# B&R Automation Studio project AriesV2 (part 2)

- acp10err-en.txt (not shown)

### ArUser.typ
```iecst
(********************************************************************
 * COPYRIGHT -- Bernecker + Rainer
 ********************************************************************
 * Library: ArUser
 * File: ArUser.typ
 * Author: B+R
 ********************************************************************
 * Data types of library ArUser
 ********************************************************************)

 TYPE
	ArUserIdentType : STRUCT
		Handle			: UDINT;
		MagicNumber		: UDINT;
	END_STRUCT;

	ArUserAsyncInternalType : STRUCT
		FBStateCtx		: ArFBStateInternalType;
		AsyFuMaCtx		: ArFBAsyFuMaInternalType;
	END_STRUCT;

	ArUserInternalType : STRUCT
		FBStateCtx		: ArFBStateInternalType;
	END_STRUCT;

END_TYPE
```

### AsGuard.var
```iecst
(********************************************************************
 * COPYRIGHT -- Bernecker + Rainer
 ********************************************************************
 * Library: AsGuard
 * File: AsGuard.var
 * Author: B+R
 ********************************************************************
 * Local variables of library AsGuard
 ********************************************************************)

(* error area 37300 - 37349 for AsGuard reserved *)

VAR CONSTANT
	guardERR_NULLPOINTER				: UINT := 37300;	(*null pointer specified*)
	guardERR_GENERAL					: UINT := 37301;	(*general license error*)
	guardERR_BUFFERSIZE					: UINT := 37302;	(*buffer too small*)
	guardERR_MEMORY						: UINT := 37303;	(*memory error*)
	guardERR_NOT_STARTED				: UINT := 37304;	(*license manager not started*)
	guardERR_ACCESS						: UINT := 37305;	(*license access error*)
	guardERR_VIOLATION					: UINT := 37306;	(*license violation*)
	guardERR_SERVICE_VIOLATION 			: UINT := 37307;	(*service mode because of license violation*)
	guardERR_CREATE_UPDATE_CONTEXT		: UINT := 37308;	(*error creating update context*)
	guardERR_CREATE_CONTEXT_FILE		: UINT := 37309;	(*error creating update context file*)
	guardERR_EXECUTE_UPDATE				: UINT := 37310;	(*error executing license update*)
	guardERR_FILE_NOT_FOUND				: UINT := 37311;	(*file not found*)
	guardERR_LIC_NOT_INITIALIZED		: UINT := 37312;	(*license not initialized*)
	guardERR_TASK						: UINT := 37313;
	guardERR_DONGLE_NOT_FOUND			: UINT := 37314;	(*specified dongle not found*)
	guardERR_CONTEXT_SIZE				: UINT := 37315;	(*wrong context size*)
	guardERR_INVALID_PARAM				: UINT := 37316;	(*invalid parameter specified*)
	guardERR_UNAVAILABLE				: UINT := 37317;	(*function unavailable*)
	guardERR_DATA_SIZE					: UINT := 37321;	(*data size invalid*)
	guardERR_LICENSE_STATUS_UNKNOWN		: UINT := 37322;	(*license status currently unknown*)

	guardBR_FIRMCODE                    : UDINT := 101652;	(*B&R firmcode*)

	guardLIC_REACT_NONE					: DWORD := 16#00;	(*no reaction*)
	guardLIC_REACT_LOGBOOK				: DWORD := 16#01;	(*in case of license violation write a message into logbook*)
	guardLIC_REACT_BLINK_CPU_LED		: DWORD := 16#02;	(*in case of license violation blink User LED*)
	guardLIC_REACT_BOOT_SERVICE			: DWORD := 16#04;	(*in case of license violation during bootup start PLC in service mode*)
	guardLIC_REACT_SERVICE				: DWORD := 16#08;	(*in case of license violation restart PLC in service mode *)

	guardREGISTER_ALWAYS				: DWORD := 1;		(*register license always*)
	guardREGISTER_IF_AVAILABLE			: DWORD := 2;		(*register license only if available*)

	guardGENERAL_OP_TIME_COUNTER 		: UDINT := 1;		(*general operating time counter*)
	guardCUSTOMER_OP_TIME_COUNTER		: UDINT := 2;		(*customer operating time counter*)
END_VAR
```

### AsHost.typ
```iecst
(********************************************************************
 * COPYRIGHT -- Bernecker + Rainer
 ********************************************************************
 * Library: AsHost
 * File: AsHost.typ
 * Author: B+R
 ********************************************************************
 * Data types of library AsHost
 ********************************************************************)

TYPE
	ASHOST_LOCAL_OBJ : STRUCT			(*internal use*)
		StateMan		: UINT;
		ErrMan			: UINT;
		Init			: UDINT;
		END_STRUCT;
END_TYPE
```

### AsOpcUac.typ
```iecst
(********************************************************************
 * COPYRIGHT -- Bernecker + Rainer
 ********************************************************************
 * Library: AsOpcUac
 * File:    AsOpcUac.typ
 * Author:  B+R
 ********************************************************************
 * Data types of library AsOpcUac
 ********************************************************************)

 TYPE
    (* Message security modes *)
	UASecurityMsgMode :
	(
    	UASecurityMsgMode_BestAvailable 	:= 0,	(* Detects best available mode the server provides (may result in no security) 	*)
	  	UASecurityMsgMode_None          	:= 1,	(* No secure communication 														*)
	  	UASecurityMsgMode_Sign          	:= 2,	(* Messages are signed to verify peer authenticity 								*)
	  	UASecurityMsgMode_SignEncrypt   	:= 3	(* Messages are signed and encrypted 											*)
	);

	(* Security policies *)
  	UASecurityPolicy :
  	(
    	UASecurityPolicy_BestAvailable  	:= 0,	(* Detects best available policy the server provides (may result in no security)	*)
    	UASecurityPolicy_None           	:= 1,	(* No secure communication (Allowed only for security mode = none)					*)
    	UASecurityPolicy_Basic128Rsa15  	:= 2,	(* RSA-PKCS-#1-V1.5-SHA1/RSA-PKCS-#1-V1.5/128-512 bit, HMAC-SHA1/AES-128-CBC/16bit	*)
    	UASecurityPolicy_Basic256       	:= 3,	(* RSA-PKCS-#1-OAEP-SHA1/RSA-OAEP/128-512 bit, HMAC-SHA1//AES-256-CBC/32bit			*)
    	UASecurityPolicy_Basic256Sha256   	:= 4	(* ???																				*)
  	);

  	(* Transport profiles to select encoding and protocol *)
  	UATransportProfile :
  	(
    	UATP_UATcp             				:= 1,	(* UA Binary over TCP								*)
    	UATP_WSHttpBinary      				:= 2,	(* Binary over HTTP			Not supported by B&R	*)
    	UATP_WSHttpXmlOrBinary 				:= 3,	(* XML/Binary over HTTP		Not supported by B&R	*)
    	UATP_WSHttpXml         				:= 4	(* XML over HTTP			Not supported by B&R	*)
  	);

  	(* Authentication token type provided for logon *)
 	UAUserIdentityTokenTtype :
 	(
 		UAUITT_Anonymous					:= 0,	(* Logon anonymously					*)
 		UAUITT_Username						:= 1,	(* Logon with user name and password 	*)
 		UAUITT_x509							:= 2	(* Logon with user certificate			*)
 	);

	(* Node identifier type *)
	UAIdentifierType :
	(
		UAIdentifierType_String 			:= 1,	(* String			*)
		UAIdentifierType_Numeric 			:= 2,	(* Numeric value	*)
		UAIdentifierType_GUID 				:= 3,	(* GUID				*)
		UAIdentifierType_Opaque				:= 4	(* ByteString		*)
	);

	(* Deadband type for monitored item sampling *)
	UADeadbandType :
	(
		UADeadbandType_None 				:= 0,	(* No deadband, each value change is sampled						*)
		UADeadbandType_Absolute 			:= 1,	(* Absolute value to exceed from last sample to make new sample		*)
		UADeadbandType_Percent				:= 2	(* Percent of EURange to exceed from last sample to make new sample	*)
	);

	UANodeClass :
	(
		UANodeClass_None 					:= 0,
		UANodeClass_Object					:= 1,
		UANodeClass_Variable 				:= 2,
		UANodeClass_Method					:= 4,
		UANodeClass_ObjectType				:= 8,
		UANodeClass_VariableType			:= 16,
		UANodeClass_ReferenceType			:= 32,
		UANodeClass_DataType				:= 64,
		UANodeClass_View					:= 128,
		UANodeClass_All						:= 255
	);

	UAAttributeId :
	(
	  	UAAI_Default						:= 0,
		UAAI_NodeId							:= 1,
		UAAI_NodeClass						:= 2,
		UAAI_BrowseName						:= 3,
		UAAI_DisplayName					:= 4,
		UAAI_Description					:= 5,
		UAAI_WriteMask						:= 6,
		UAAI_UserWriteMask					:= 7,
		UAAI_IsAbstract						:= 8,
		UAAI_Symmetric						:= 9,
		UAAI_InverseName					:= 10,
		UAAI_ContainsNoLoops				:= 11,
		UAAI_EventNotifier					:= 12,
		UAAI_Value							:= 13,
		UAAI_DataType						:= 14,
		UAAI_ValueRank						:= 15,
		UAAI_ArrayDimensions				:= 16,
		UAAI_AccessLevel					:= 17,
		UAAI_UserAccessLevel				:= 18,
		UAAI_MinimumSamplingInterval		:= 19,
		UAAI_Historizing					:= 20,
		UAAI_Executable						:= 21,
		UAAI_UserExecutable					:= 22
	);

	UAConnectionStatus :
	(
		UACS_Connected						:= 0,
		UACS_ConnectionError				:= 1,
		UACS_Shutdown						:= 2
	);

	UAServerState :
	(
		UASS_Running						:= 0,
		UASS_Failed							:= 1,
		UASS_NoConfiguration				:= 2,
		UASS_Suspended						:= 3,
		UASS_Shutdown						:= 4,
		UASS_Test							:= 5,
		UASS_CommunicationFault				:= 6,
		UASS_Unknown              			:= 7
	);

	UAVariantType :
	(										(* Kind of the variant data *)
		UAVariantType_Null					:= 0,	(* No data *)
		UAVariantType_Boolean				:= 1,	(* Data in element Boolean *)
		UAVariantType_SByte					:= 2,	(* Data in element SByte *)
		UAVariantType_Byte					:= 3,	(* Data in element Byte *)
		UAVariantType_Int16					:= 4,	(* Data in element Int16 *)
		UAVariantType_UInt16				:= 5,	(* Data in element UInt16 *)
		UAVariantType_Int32					:= 6,	(* Data in element Int32 *)
		UAVariantType_UInt32				:= 7,	(* Data in element UInt32 *)
		UAVariantType_Int64					:= 8,	(* Data in element Int64 *)
		UAVariantType_UInt64				:= 9,	(* Data in element UInt64 *)
		UAVariantType_Float					:= 10,	(* Data in element Float *)
		UAVariantType_Double				:= 11,	(* Data in element Double *)
		UAVariantType_String				:= 12,	(* Data in element String *)
		UAVariantType_DateTime				:= 13,	(* Data in element DateTime *)
		UAVariantType_Guid					:= 14,	(* Guid data in element String *)
		UAVariantType_ByteString			:= 15,	(* Byte string in element String *)
		UAVariantType_XmlElement			:= 16,	(* XML data in element String *)
		UAVariantType_NodeId				:= 17,	(* Data in element NodeId *)
		UAVariantType_ExpandedNodeId		:= 18,	(* Data in element ExpandedNodeId *)
		UAVariantType_StatusCode			:= 19,	(* Status code in element UInt32 *)
		UAVariantType_QualifiedName			:= 20,	(* Data in element QualifiedName *)
		UAVariantType_LocalizedText			:= 21	(* Data in element LocalizedText *)
	);

   	UAUserIdentityToken : STRUCT
		UserIdentityTokenType	: UAUserIdentityTokenTtype;
		TokenParam1 			: STRING[255];
		TokenParam2				: STRING[255];
	END_STRUCT;

 	UASessionConnectInfo : STRUCT
 	  	SessionName   			: STRING[255];
 	  	ApplicationName   		: STRING[255];
 	  	SecurityMsgMode   		: UASecurityMsgMode;
    	SecurityPolicy   		: UASecurityPolicy;
		CertificateStore		: STRING[255];
		ClientCertificateName	: STRING[255];
		ServerUri				: STRING[255];
		CheckServerCertificate	: BOOL;
    	TransportProfile 		: UATransportProfile;
    	UserIdentityToken		: UAUserIdentityToken;
		VendorSpecificParameter	: STRING[255];
    	SessionTimeout   		: TIME;
    	MonitorConnection		: TIME;
    	LocaleIDs				: ARRAY[0..4] OF STRING[6];
	END_STRUCT;

	(* Node identifier used to address nodes on the server *)
  	UANodeID : STRUCT
		NamespaceIndex			: UINT;							(* Index of the namespace which contains the node			*)
		Identifier 				: STRING[255];					(* Node identifier according to the identifier types format *)
		IdentifierType			: UAIdentifierType; 			(* String, Numeric, GUID, ByteString						*)
	END_STRUCT;

	(* Settings for data item monitoring *)
	UAMonitoringSettings : STRUCT
		SamplingInterval		: TIME;							(* Time in ms 															*)
		DeadbandType			: UADeadbandType; 				(* Deadband type which applies to deadband value						*)
		Deadband				: REAL; 						(* Deadband value, semantics depending on DeadbandType 					*)
	END_STRUCT;

	(* Settings for data item monitoring *)
	UAMonitoringParameters : STRUCT
		SamplingInterval		: TIME;							(* Time in ms 															*)
		QueueSize				: UINT;							(* Size of the server sided queue to collect value changes				*)
		DiscardOldest			: BOOL;							(* True to discard oldest on queue overflow or newest otherwise			*)
		DeadbandType			: UADeadbandType; 				(* Deadband type which applies to deadband value						*)
		Deadband				: REAL; 						(* Deadband value, semantics depending on DeadbandType 					*)
	END_STRUCT;

	UALocalizedText : STRUCT
		Locale					: STRING[6];
		Text					: STRING[255];
	END_STRUCT;

	UANodeInfo : STRUCT
		AccessLevel 			: BYTE;
		ArrayDimension			: ARRAY[0..MAX_INDEX_ARRAYDIMENSION] OF UDINT;
		BrowseName				: STRING[255];
		ContainsNoLoops 		: BOOL;
		DataType				: UANodeID;
		Description				: UALocalizedText;
		DisplayName				: UALocalizedText;
		EventNotifier			: BYTE;
		Executable				: BOOL;
		Historizing				: BOOL;
		InverseName				: STRING[255];
		IsAbstract				: BOOL;
		MinimumSamplingInterval	: TIME;
		NodeClass				: UANodeClass;
		NodeID					: UANodeID;
		Symmetric				: BOOL;
		UserAccessLevel			: BYTE;
		UserExecutable			: BOOL;
		UserWriteMask			: UDINT;
		ValueRank				: DINT;
		WriteMask				: UDINT;
	END_STRUCT;

	UAIndexRange : STRUCT
		StartIndex				: UINT;
		EndIndex 				: UINT;
	END_STRUCT;

	UANodeAdditionalInfo : STRUCT
		AttributeId				: UAAttributeId;
		IndexRangeCount			: UINT;
		IndexRange 				: ARRAY[0..MAX_INDEX_INDEXRANGE] OF UAIndexRange;
	END_STRUCT;

	(* Method argument used to supply the input and receive the output argument values for method calls *)
	UAMethodArgument : STRUCT
		Name					: STRING[64];		(* Name of the method argument								*)
		Value					: STRING[255];		(* Source/Destination variable name for the argument value	*)
	END_STRUCT;

	UAExpandedNodeID : STRUCT 	(* Expanded node identfier type *)
		NodeId					: UANodeID;
		NamespaceUri			: STRING[255];
		ServerIndex				: UDINT;
	END_STRUCT;

	UAQualifiedName : STRUCT	(* Qualified name type *)
		NamespaceIndex			: UINT;
		Name					: STRING[255];
	END_STRUCT;

	UARelativePathElement : STRUCT
	    ReferenceTypeId			: UANodeID;
		IsInverse				: BOOL;
		IncludeSubTypes			: BOOL;
		TargetName				: UAQualifiedName;
	END_STRUCT;

	UARelativePath : STRUCT
	    NoOfElements			: DWORD;
		Elements				: ARRAY[0..MAX_INDEX_RELATIVEPATH] OF UARelativePathElement;
	END_STRUCT;

	UADataValue : STRUCT		(* Additional informations about data value *)
		Valid 					: BOOL;
		Reserved				: ARRAY[0..2]OF USINT;
		StatusCode				: UDINT;
		SourceTimestamp			: DATE_AND_TIME;
		ServerTimestamp			: DATE_AND_TIME;
	END_STRUCT;

	UAVariantData : STRUCT		(* Standard type for variant data *)
		VariantType				: UAVariantType;
		Boolean					: BOOL;
		SByte					: SINT;
		Byte					: USINT;
		Int16					: INT;
		UInt16					: UINT;
		Int32					: DINT;
		UInt32					: UDINT;
		Float					: REAL;
		Double					: LREAL;
		DateTime				: DATE_AND_TIME;
		String					: STRING[255];
		NodeId					: UANodeID;
		ExpandedNodeId			: UAExpandedNodeID;
		QualifiedName			: UAQualifiedName;
		LocalizedText			: UALocalizedText;
		DataValue				: UADataValue;
	END_STRUCT;

	UARange : STRUCT			(* Range for a value *)
		Low						: LREAL;
		High					: LREAL;
	END_STRUCT;

	UAEUInformation : STRUCT 	(* Information about the engineering units *)
		NamespaceUri			: STRING[255];
		UnitId					: DINT;
		DisplayName				: UALocalizedText;
		Description				: UALocalizedText;
	END_STRUCT;

	UATimeZoneData : STRUCT		(* Information about time zone *)
		TimeOffset				: INT;	(* Offset in minutes from UTC *)
		DaylightSaving			: BOOL;	(* Offset includes the DST *)
	END_STRUCT;

END_TYPE
```

### AsSafety.typ
```iecst
(********************************************************************
 * COPYRIGHT -- Bernecker + Rainer
 ********************************************************************
 * Library: AsSafety
 * File: AsSafety.typ
 * Author: B&R
 * Created: May 25, 2012
 ********************************************************************
 * Data types of library AsSafety
 ********************************************************************)

TYPE
	RemoteControlCmdTypeV1 : 	STRUCT  (*remote control command structure*)
		Version : UINT; (*used version*)
		Command : UINT; (*command*)
		Number : UINT; (*actual number*)
		Data : UINT; (*data*)
		Password : STRING[16]; (*password*)
		NewPassword : STRING[16]; (*new password*)
	END_STRUCT;
	DownloadCmdMaOpTypeV1 : 	STRUCT  (*machine options command structure*)
		Version : UINT; (*used version*)
		Password : STRING[16]; (*password*)
		UDID_Low : UDINT; (*UDID low from SafeLOGIC*)
		UDID_High : UINT; (*UDID high from SafeLOGIC*)
		Unlock : USINT; (*unlock data*)
		pDeviceListInput : UDINT; (*pointer to device list*)
		NumberDevicesInput : UINT; (*number of devices*)
		pMachineOptionsInput : UDINT; (*pointer to bit machine options*)
		pModuleFlagsInput : UDINT; (*pointer to module flags*)
		pAcknMachineOptions : UDINT; (*pointer to acknowledge information*)
		pDeviceListOutput : UDINT; (*pointer to device list from SafeLOGIC*)
		NumberDevicesOutput : UINT; (*number of devices from SafeLOGIC*)
		pMachineOptionsOutput : UDINT; (*pointer to bit machine options from SafeLOGIC*)
		pModuleFlagsOutput : UDINT; (*pointer to module flags from SafeLOGIC*)
	END_STRUCT;
	DownloadDeviceTypeV1 : 	STRUCT  (*safety device*)
		SADR : UINT; (*safety address*)
		UDID_Low : UDINT; (*UDID low*)
		UDID_High : UINT; (*UDID high*)
	END_STRUCT;
	ConfigurationDeviceTypeV1 : 	STRUCT  (*safety device from SafeLOGIC*)
		SADR : UINT; (*safety address*)
		UDID : ARRAY[0..5]OF USINT; (*UDID*)
	END_STRUCT;
	ConfigurationBitOptionsTypeV1 : 	STRUCT  (*bit machine options*)
		BitData : ARRAY[0..63]OF USINT; (*bit array*)
	END_STRUCT;
	ConfigurationModuleFlagsTypeV1 : 	STRUCT  (*module flags*)
		Optional : ARRAY[0..127]OF USINT; (*optional*)
		Startup : ARRAY[0..127]OF USINT; (*startup*)
		NotPresent : ARRAY[0..127]OF USINT; (*not present*)
	END_STRUCT;
	DownloadCmdExtMaOpTypeV1 : 	STRUCT  (*extended machine options command structure*)
		Version : UINT; (*used version*)
		Password : STRING[16]; (*password*)
		UDID_Low : UDINT; (*UDID low*)
		UDID_High : UINT; (*UDID high*)
		Unlock : USINT; (*unlock data*)
		pIntDataInput : UDINT; (*pointer to INT data*)
		NumberIntInput : UINT; (*number of INT channels*)
		pUintDataInput : UDINT; (*pointer to UINT data*)
		NumberUintInput : UINT; (*number of UINT channels*)
		pDintDataInput : UDINT; (*pointer to DINT data*)
		NumberDintInput : UINT; (*number of DINT channels*)
		pUdintDataInput : UDINT; (*pointer to UDINT data*)
		NumberUdintInput : UINT; (*number of UDINT channels*)
		pAcknMachineOptions : UDINT; (*pointer to acknowledge information*)
		pIntDataOutput : UDINT; (*pointer to INT data from SafeLOGIC*)
		NumberIntOutput : UINT; (*number of INT channels from SafeLOGIC*)
		pUintDataOutput : UDINT; (*pointer to UINT data from SafeLOGIC*)
		NumberUintOutput : UINT; (*number of UINT channels from SafeLOGIC*)
		pDintDataOutput : UDINT; (*pointer to DINT data from SafeLOGIC*)
		NumberDintOutput : UINT; (*number of DINT channels from SafeLOGIC*)
		pUdintDataOutput : UDINT; (*pointer to UDINT data from SafeLOGIC*)
		NumberUdintOutput : UINT; (*number of UDINT channels from SafeLOGIC*)
	END_STRUCT;
	ConfigurationIntOptionsTypeV1 : 	STRUCT  (*INT machine options*)
		ID : UINT; (*id*)
		Value : INT; (*value*)
	END_STRUCT;
	ConfigurationUintOptionsTypeV1 : 	STRUCT  (*UINT machine options*)
		ID : UINT; (*id*)
		Value : UINT; (*value*)
	END_STRUCT;
	ConfigurationDintOptionsTypeV1 : 	STRUCT  (*DINT machine options*)
		ID : UINT; (*id*)
		Value : DINT; (*value*)
	END_STRUCT;
	ConfigurationUdintOptionsTypeV1 : 	STRUCT  (*UDINT machine options*)
		ID : UINT; (*id*)
		Value : UDINT; (*value*)
	END_STRUCT;
	DownloadCmdTableTypeV1 : 	STRUCT  (*table command structure*)
		Version : UINT; (*used version*)
		Password : STRING[16]; (*password*)
		UDID_Low : UDINT; (*UDID low*)
		UDID_High : UINT; (*UDID high*)
		Unlock : USINT; (*unlock data*)
		pTableDataInput : UDINT; (*pointer to table data*)
		NumberTablesInput : UINT; (*number of tables*)
		pTableDataOutput : UDINT; (*pointer to table data from SafeLOGIC*)
		NumberTablesOutput : UINT; (*number of tables from SafeLOGIC*)
	END_STRUCT;
	DownloadCmdAddParaTypeV1 : 	STRUCT  (*additional paramater command structure*)
		Version : UINT; (*used version*)
		Password : STRING[16]; (*password*)
		UDID_Low : UDINT; (*UDID low*)
		UDID_High : UINT; (*UDID high*)
		Unlock : USINT; (*unlock data*)
		pParaListInput : UDINT; (*pointer to additional parameter data*)
		NumberParaSetsInput : UINT; (*number of parameter sets*)
		pParaDataOutput : UDINT; (*pointer to additional parameter data from SafeLOGIC*)
		NumberParaSetsOutput : UINT; (*number of parameter sets from SafeLOGIC*)
	END_STRUCT;
	DownloadTableTypeV1 : 	STRUCT  (*table data*)
		Device : STRING[80]; (*device for file*)
		File : STRING[80]; (*file name*)
	END_STRUCT;
	ConfigurationTableTypeV1 : 	STRUCT  (*table data from SafeLOGIC*)
		ID : UINT; (*table id*)
		Type : USINT; (*table type*)
		NumberOfCRCs : UINT; (*number of CRCs*)
		pCRCData : UDINT; (*pointer to CRC values*)
	END_STRUCT;
	DownloadAddParaTypeV1 : 	STRUCT  (*additional parameter data*)
		SADR : UINT; (*safety address*)
		ID : USINT; (*id*)
		pParaData : UDINT; (*pointer to additional parameter data*)
		Length : UDINT; (*length*)
		pAcknAddPara : UDINT; (*pointer to acknowledge information*)
	END_STRUCT;
	ConfigurationAddParaTypeV1 : 	STRUCT  (*additional parameter data from SafeLOGIC*)
		SADR : UINT; (*safety address*)
		ID : USINT; (*id*)
		pParaData : UDINT; (*pointer to additional parameter data*)
		Length : UDINT; (*length*)
		CRC : UDINT; (*CRC*)
		Timestamp : UDINT; (*timestamp*)
	END_STRUCT;
	DownloadCmdApplicationTypeV1 : 	STRUCT  (*application command structure*)
		Version : UINT; (*used version*)
		Password : STRING[16]; (*password*)
		UDID_Low : UDINT; (*UDID low*)
		UDID_High : UINT; (*UDID high*)
		ApplicationID : UINT; (*application id*)
		Device : STRING[80]; (*device for file*)
		File : STRING[80]; (*file name*)
		Unlock : USINT; (*unlock application*)
	END_STRUCT;
	ConfigurationCmdMaOpTypeV1 : 	STRUCT  (*machine options from SafeLOGIC command structure*)
		Version : UINT; (*used version*)
		Password : STRING[16]; (*password*)
		pDeviceListOutput : UDINT; (*pointer to device list from SafeLOGIC*)
		NumberDevicesOutput : UINT; (*number of devices from SafeLOGIC*)
		pMachineOptionsOutput : UDINT; (*pointer to bit machine options from SafeLOGIC*)
		pModuleFlagsOutput : UDINT; (*pointer to module flags from SafeLOGIC*)
	END_STRUCT;
	ConfigurationCmdExtMaOpTypeV1 : 	STRUCT  (*extended machine options from SafeLOGIC command structure*)
		Version : UINT; (*used version*)
		Password : STRING[16]; (*password*)
		pIntDataOutput : UDINT; (*pointer to INT data from SafeLOGIC*)
		NumberIntOutput : UINT; (*number of INT channels from SafeLOGIC*)
		pUintDataOutput : UDINT; (*pointer to UINT data from SafeLOGIC*)
		NumberUintOutput : UINT; (*number of UINT channels from SafeLOGIC*)
		pDintDataOutput : UDINT; (*pointer to DINT data from SafeLOGIC*)
		NumberDintOutput : UINT; (*number of DINT channels from SafeLOGIC*)
		pUdintDataOutput : UDINT; (*pointer to UDINT data from SafeLOGIC*)
		NumberUdintOutput : UINT; (*number of UDINT channels from SafeLOGIC*)
	END_STRUCT;
	ConfigurationCmdTableTypeV1 : 	STRUCT  (*table data from SafeLOGIC command structure*)
		Version : UINT; (*used version*)
		Password : STRING[16]; (*password*)
		pTableDataOutput : UDINT; (*pointer to table data from SafeLOGIC*)
		NumberTablesOutput : UINT; (*number of tables from SafeLOGIC*)
	END_STRUCT;
	ConfigurationCmdAddParaTypeV1 : 	STRUCT  (*additional parameter data from SafeLOGIC command structure*)
		Version : UINT; (*used version*)
		Password : STRING[16]; (*password*)
		pParaDataOutput : UDINT; (*pointer to additional parameter data from SafeLOGIC*)
		NumberParaSetsOutput : UINT; (*number of parameter sets from SafeLOGIC*)
	END_STRUCT;
	RemoteControlStatusTypeV1 : 	STRUCT  (*remote control status from SafeLOGIC*)
		Command : UINT; (*last received command*)
		Number : UINT; (*running number of last received command*)
		Status : UINT; (*status of command*)
		State : UINT; (*state of the last ENTER command*)
		EnterData : UINT; (*last received ENTER command that was correct executed*)
		EnterNumber : UINT; (*running number of the last received ENTER command*)
		EnterExecuteStatus : UINT; (*state of the last received ENTER command*)
		SafeOSState : USINT; (*status of the safety application*)
		SafeKEYChanged : USINT; (*SafeKEY has been exchanged*)
		LedTestActive : USINT; (*LED test active*)
		Scanning : USINT; (*module scan active*)
		openSAFETYstate : USINT; (*status of openSAFETY stack*)
		FailSafe : USINT; (*Fail-Safe status*)
		NumberOfMissingModules : UINT; (*number of missing modules*)
		NumberOfUDIDMismatches : UINT; (*number of mismatched modules*)
		NumberOfDifferentFirmware : UINT; (*number of modules with different firmware*)
		SADR : ARRAY[0..100]OF UINT; (*safety address array*)
		MissingModules : ARRAY[0..15]OF USINT; (*missing modules array*)
		UDIDMismatches : ARRAY[0..15]OF USINT; (*udid mismatch array*)
		DifferentFirmware : ARRAY[0..15]OF USINT; (*different firmware array*)
	END_STRUCT;
	DownloadAcknMaOpTypeV1 : 	STRUCT  (*acknowledge bit machine options structure*)
		AcknBitOptions : ARRAY[0..63]OF USINT; (*acknowledge bit*)
	END_STRUCT;
	DownloadAcknAddParaTypeV1 : 	STRUCT  (*acknowledge bit additional parameter*)
		AcknBitAddPara : ARRAY[0..63]OF USINT; (*acknowledge bit*)
	END_STRUCT;
	DownloadAcknExtMaOpTypeV1 : 	STRUCT  (*acknowledge extended machine options structure*)
		AcknIntOptions : ARRAY[0..63]OF BOOL; (*acknowledge INT*)
		AcknUintOptions : ARRAY[0..63]OF BOOL; (*acknowledge UINT*)
		AcknDintOptions : ARRAY[0..63]OF BOOL; (*acknowledge DINT*)
		AcknUdintOptions : ARRAY[0..63]OF BOOL; (*acknowledge UDINT*)
	END_STRUCT;
END_TYPE
```

### AsSafety.var
```iecst
(********************************************************************
 * COPYRIGHT -- Bernecker + Rainer
 ********************************************************************
 * Library: AsSafety
 * File: AsSafety.var
 * Author: B&R
 * Created: May 25, 2012
 ********************************************************************
 * Constants of library AsSafety
 ********************************************************************)
VAR CONSTANT
	safeVERSION_R107 : UINT := 16#107; (*safety release version - for 1.7 or higher*)
	safeDATA_TYPE_MAOP : UINT := 16#100; (*download type for machine options *)
	safeDATA_TYPE_EXTMAOP : UINT := 16#200; (*download type for extended machine options *)
	safeDATA_TYPE_TABLE : UINT := 16#300; (*download type for table objects *)
	safeDATA_TYPE_ADDPARA : UINT := 16#400; (*download type for additional parameter*)
	safeCMD_ENTER : UINT := 16#100; (*enter command*)
	safeCMD_STATUS : UINT := 16#200; (*status command*)
	safeCMD_STATUS_SL : UINT := 16#0000; (*read back status*)
	safeCMD_N_UDID_ACKN : UINT := 16#20; (*acknowledge N modules*)
	safeCMD_4_UDID_ACKN : UINT := 16#30; (*acknowledge 4 modules*)
	safeCMD_3_UDID_ACKN : UINT := 16#40; (*acknowledge 3 modules*)
	safeCMD_2_UDID_ACKN : UINT := 16#50; (*acknowledge 2 modules*)
	safeCMD_1_UDID_ACKN : UINT := 16#60; (*acknowledge 1 module*)
	safeCMD_FW_ACKN : UINT := 16#100; (*acknowledge firmware*)
	safeCMD_SK_XCHG : UINT := 16#200; (*acknowledge SafeKEY*)
	safeCMD_TEST : UINT := 16#1000; (*LED test*)
	safeCMD_SCAN : UINT := 16#2000; (*scan*)
	safeCMD_SK_PW : UINT := 16#5000; (*change password*)
	safeCMD_SK_FORMAT : UINT := 16#6000; (*format SafeKEY*)
	safeCMD_RESET : UINT := 16#7000; (*reset SafeLOGIC*)
	safeCMD_CLEAR_DATA : UINT := 16#8000; (*clear additonal downloaded data*)
	safeERR_VERSION : UINT := 36100; (*error wrong version for command structure*)
	safeERR_PW_LENGTH : UINT := 36101; (*error wrong password length*)
	safeERR_UDID : UINT := 36102; (*error no UDID*)
	safeERR_ALLOC_MEM : UINT := 36103; (*error allocating memory*)
	safeERR_INTERNAL_ERROR : UINT := 36104; (*internal error*)
	safeERR_TIMEOUT : UINT := 36105; (*error connection timeout*)
	safeERR_RC_CMD : UINT := 36106; (*error wrong command*)
	safeERR_RC_ENTER_DATA : UINT := 36107; (*error wrong data for ENTER command*)
	safeERR_RC_ENTER_PW : UINT := 36108; (*error no password for command*)
	safeERR_RC_ENTER_SK_PW : UINT := 36109; (*error no new password for command*)
	safeERR_RC_STATUS_DATA : UINT := 36110; (*error wrong data for STATUS command*)
	safeERR_RC_DATA_LENGTH : UINT := 36111; (*error worng length for status data*)
	safeERR_DL_NO_PASSWORD : UINT := 36112; (*error no password for download*)
	safeERR_DL_PROTOCOL : UINT := 36113; (*error protocol version for download*)
	safeERR_DL_FILE_OPEN : UINT := 36114; (*error file open*)
	safeERR_DL_FILE_INVALID : UINT := 36115; (*error file invalid*)
	safeERR_DL_FILE_TOO_BIG : UINT := 36116; (*error file too big*)
	safeERR_DL_WRITE : UINT := 36117; (*error write*)
	safeERR_DL_STREAM : UINT := 36118; (*error stream*)
	safeERR_DL_CHECKSUM : UINT := 36119; (*error checksum*)
	safeERR_DL_UDID : UINT := 36120; (*error UDID doesn't match*)
	safeERR_DL_WRONG_FILE_SIZE : UINT := 36121; (*error wrong file size*)
	safeERR_DL_NO_RIGHTS_TO_WRITE : UINT := 36122; (*error wrong password*)
	safeERR_DL_UNLOCK_FILE_INFO : UINT := 36123; (*error file info*)
	safeERR_DL_UNLOCK_READ : UINT := 36124; (*error unlock read*)
	safeERR_DL_UNLOCK_WRITE : UINT := 36125; (*error unlock write*)
	safeERR_DL_STATIC_UNLOCK : UINT := 36126; (*error static unlock*)
	safeERR_DL_COMPARE_FAILED : UINT := 36127; (*error data compare failed*)
	safeERR_DLDATA_TYPE_ERR : UINT := 36128; (*error data type for download*)
	safeERR_DLDATA_ERR_DATA : UINT := 36129; (*error data for download*)
	safeERR_COT_TYPE_ERR : UINT := 36130; (*error data type for upload*)
	safeERR_COT_READING_FILE : UINT := 36131; (*error reading file*)
END_VAR
```

### GmcManager.typ
```iecst
TYPE
	(*Enum types*)

	MCBufferModeEnum :
	(
		mcABORTING, (*Default mode with no buffering. The function block aborts an active movement. The buffer is cleared.*)
		mcBUFFERED 	(*The movement is started as soon as the previous movement is completed. No smoothing is applied.*)
	);

	MCCoordinateSystemEnum :
	(
		mcACS := 0,	(*Axis coordinate system*)
		mcMCS := 1,	(*Machine coordinate system*)
		mcPCS := 2,	(*Product coordinate system*)
		mcSCS1 := 3,	(*System coordinate system 1*)
		mcSCS2 := 4,	(*System coordinate system 2*)
		mcSCS3 := 5,	(*System coordinate system 3*)
		mcSCS4 := 6,	(*System coordinate system 4*)
		mcSCS5 := 7,	(*System coordinate system 5*)
		mcJACS := 100	(*Joint axis coordinate system*)
	);

	MCDirectionEnum :
	(
		mcDIR_POSITIVE,	(*positive direction*)
		mcDIR_NEGATIVE,	(*negative direction*)
		mcDIR_CURRENT,	(*current direction*)
		mcDIR_SHORTEST_WAY,		(*shortest way*)
		mcDIR_EXCEED_PERIOD := 8,	(*exceed period*)
		mcDIR_UNDEFINED	(*undefined direction*)
	);

	MCErrorCommandEnum :
	(
		mcWARNING_CMD := 0, (*a warning is generated*)
		mcERROR_CMD, (*Generates an error*)
		mcERROR_STOP_CMD, (*Generates an error and stops.*)
		mcERROR_STOP_CTRL_OFF_CMD, (*an axis error is generated on the drive, any active movement is aborted and the controller is switched off*)
		mcERROR_V_STOP_CTRL_OFF_CMD (*an axis error is generated on the drive, any active movement is ended with a speed ramp and controller is switched off*)
	);

	MCExecutionModeEnum :
	(
		mcEM_IMMEDIATELY,	(*The function is executed immediately.*)
		mcEM_QUEUED			(*The function is executed with a buffer.*)
	);

	MCGroupOperationModeEnum :
	(
		mcOM_M1_STOP, (*Optional stop*)
		mcOM_FEED_FORWARD, (*Feed forward*)
		mcOM_OPTMOT, (*Jerk-limiting trajectory planner*)
		mcOM_SAVE_RESTARTDATA (*Save data to restart a program*)
	);

	MCUnloadProgramModeEnum :
	(
		mcUPRG_NAME, (*Unload program by name*)
		mcUPGR_ALL (*Unload all programs*)
	);

	MCHomingModeEnum :
	(
		mcHOMING_DIRECT := 0,			(*Direct homing*)
		mcHOMING_SWITCH_GATE,			(*Homing with reference gate*)
		mcHOMING_ABSOLUTE_SWITCH,		(*Performs homing with absolute reference switch*)
		mcHOMING_LIMIT_SWITCH := 4,	    (*Homing with hardware limit switch*)
		mcHOMING_ABSOLUTE,				(*Homing by setting the homing offset*)
		mcHOMING_DCM := 7,				(*Homing using interval-encoded reference marks*)
		mcHOMING_BLOCK_TORQUE := 9,	    (*Performs homing to mechanical limit, torque as criteria*)
		mcHOMING_BLOCK_LAG_ERROR := 10,	(*Performs homing to mechanical limit, lag error as criteria*)
		mcHOMING_ABSOLUTE_CORRECTION := 133, (*Homing by setting the homing offset with counting range correction*)
		mcHOMING_DCM_CORRECTION := 135,	(*Homing using distance-coded reference marks with counting range correction*)
		mcHOMING_DEFAULT := 140,		(*Applies all parameters from the configuration*)
		mcHOMING_INIT,					(*init*)
		mcHOMING_RESTORE_POSITION		(*Restores position from permanent memory*)
	);

	MCHomingOrderSourceEnum :
	(
		mcHO_CONFIGURATION := 0,	(*Uses the homing order configured in the configuration*)
		mcHO_FUNCTIONBLOCK			(*Uses the homing order configured in the function block*)
	);

	MCInterpolationModeEnum :
	(
		mcIPLM_OFF,						(*interpolation off*)
		mcIPLM_LINEAR,					(*linear interpolation*)
		mcIPLM_QUADRATIC,				(*quadratic interpolation*)
		mcIPLM_QUADRATIC_NO_OVERSHOOT	(*quadratic interpolation without overshoot*)
	);

	MCOverrideEnum :
	(
		mcOVERRIDE_VELOCITY,			(*Speed override*)
		mcOVERRIDE_VELOCITY_AXIS,		(*Axis speed override*)
		mcOVERRIDE_ACCELERATION,		(*Acceleration override*)
		mcOVERRIDE_ACCELERATION_AXIS,	(*Axis acceleration override*)
		mcOVERRIDE_JERK,				(*Jerk override*)
		mcOVERRIDE_FEEDRATE := 10,		(*Feed override*)
		mcOVERRIDE_RAPID,				(*Rapid motion override*)
		mcOVERRIDE_SPINDLE,				(*Spindle override*)
		mcOVERRIDE_TIMESTRETCH := 20	(*Time stretch override*)
	);

	MCPlcopenParameterEnum :
	(
		mcPAR_COMMANDED_AX_POSITION := 1, 	(*Commanded position*)
		mcPAR_SW_LIMIT_POSITIVE,		(*Positive software limit*)
		mcPAR_SW_LIMIT_NEGATIVE,		(*Negative software limit*)
		mcPAR_ENABLE_LIMIT_POSITIVE,	(*Enable positive software limit switch*)
		mcPAR_ENABLE_LIMIT_NEGATIVE,	(*Enable negative software limit switch*)
		mcPAR_ENABLE_POS_LAG_MONITORING,	(*Enable monitoring of position lag*)
		mcPAR_MAX_AX_POSITION_LAG,		(*Maximum position lag*)
		mcPAR_MAX_AX_VELOCITY_SYSTEM,	(*Maximum velocity of the axis in the system*)
		mcPAR_MAX_AX_VELOCITY_APPL,		(*Maximum velocity of the axis in the application*)
		mcPAR_ACTUAL_AX_VELOCITY,  		(*Actual velocity of the axis*)
		mcPAR_COMMANDED_AX_VELOCITY,	(*Commanded velocity*)
		mcPAR_MAX_AX_ACCELERATION_SYSTEM,	(*Maximum acceleration of the axis in the system*)
		mcPAR_MAX_AX_ACCELERATION_APPL,	(*Maximum acceleration of the axis in the application*)
		mcPAR_MAX_AX_DECELERATION_SYSTEM,	(*Maximum deceleration of the axis in the system*)
		mcPAR_MAX_AX_DECELERATION_APPL,	(*Maximum deceleration of the axis in the application*)
		mcPAR_MAX_AX_JERK,			(*Maximum jerk of the axis*)
		mcPAR_AX_PERIOD := 1008,    (*Period of the axis*)
		mcPAR_HOMING_OFFSET := 1019, 	(*Homing offset of the axis*)
		mcPAR_AX_MEASUREMENT_RESOLUTION := 1020  (*Measurement resolution of the axis*)
	);

	MCNetworkTypeEnum :
	(
		mcNETWORK_POWERLINK	(*ETHERNET POWERLINK protocol*)
	);

	MCPrgAxesReposTypeEnum :
	(
		mcPRGRP_SINGLE_AXIS,			(*Single axis*)
		mcPRGRP_PROGRAM,				(*Program*)
		mcPRGRP_SINGLE_AXIS_AUTOMATIC	(*Single axis automatic*)
	);

	MCPrgInfoInterruptEnum :
	(
		mcINTERRUPT_NOT_INTERRUPTED,	(*The program has not been interrupted.*)
		mcINTERRUPT_SINGLESTEP,			(*The program has been interrupted by activation of single-step mode.*)
		mcINTERRUPT_FB,					(*The program has been interrupted by the "MC_GroupInterrupt" function block.*)
		mcINTERRUPT_INTERPRETER,		(*The program has been interrupted by an interpreter halt (G170).*)
		mcINTERRUPT_MFUNCTION,			(*The program has been interrupted by a blocking M-code.*)
		mcINTERRUPT_PROGRAM				(*The program has been interrupted by a programmed command.*)
	);

	MCPrgInfoModeEnum :
	(
		mcPRGIM_LIVE,		(*Live data*)
		mcPRGIM_ABORT_POINT (*Abortpoint data*)
	);

	MCRestartModeEnum :
	(
	   	mcRSM_ABORT_LINE,		(*Restart at abort line*)
		mcRSM_PATH_DISTANCE,	(*Restart at path distance*)
		mcRSM_BLOCK_NUMBER,		(*Restart at block number*)
		mcRSM_LINE_NUMBER,		(*Restart at line number*)
		mcRSM_TOOL_NUMBER,		(*Restart at tool number*)
		mcRSM_LABEL				(*Restart at label*)
	);

	MCRestartPhaseEnum :
	(
		mcRSP_INACTIVE,
		mcRSP_VALIDATE_PLAY_BACK_DATA,
		mcRSP_WAIT_START_AXES_REPOS,
		mcRSP_AXES_REPOSITIONING,
		mcRSP_WAIT_RESTART_PROGRAM,
		mcRSP_RUN_PROGRAM,
		mcRSP_PROGRAM_FINISHED
	);

	MCPrgStartModeEnum :
	(
		mcPRGSM_NON_MODAL,		(*Non Modal*)
		mcPRGSM_MODAL,		(*Modal*)
		mcPRGSM_RESTART		(*Restart*)
	);

	MCPrgStartPointEnum :
	(
		mcPRGSP_STANDARD,		(*Standard*)
		mcPRGSP_BLOCK_NUMBER,	(*Block Number*)
		mcPRGSP_ABORT_LINE,	(*Abort Line*)
		mcPRGSP_ABORT_POINT,	(*Abort Point*)
		mcPRGSP_PATH_DISTANCE,	(*Path Distance*)
		mcPRGSP_LINE_NUMBER	(*Line Number*)
	);

	MCPrgPhaseEnum :
	(
		mcPRGPH_INACTIVE,					(*Inactive*)
		mcPRGPH_SIMULATION_RUN,			(*Simulation run is active*)
		mcPRGPH_WAIT_FOR_AXES_REPOS,		(*Waiting for axes repositioning*)
		mcPRGPH_AXES_REPOS,				(*Axes repositioning is active*)
		mcPRGPH_WAIT_FOR_REAL_RUN,			(*Waiting for real run*)
		mcPRGPH_REAL_RUN					(*Real run is active*)
	);

	MCSimulationCommandEnum :
	(
		mcSIMULATION_SW_OFF,	(*simulation off*)
		mcSIMULATION_SW_ON		(*motor simulation*)
	);

	MCSwitchEnum :
	(
		mcSWITCH_STATE_OFF,		(*off*)
		mcSWITCH_STATE_ON		(*on*)
	);

	MCTransitionModeEnum :
	(
		mcTM_NONE		(*No transition is applied*)
	);

	MCValueSourceEnum :
	(
		mcVALUE_SET, 					(*Set position is used*)
		mcVALUE_ACTUAL,					(*Actual position is used*)
		mcVALUE_SET_AXIS_UNITS,			(*Set position in axis units is used*)
		mcVALUE_ACTUAL_AXIS_UNITS,		(*Actual position in axis units is used*)
		mcVALUE_AUTOMATIC_SELECTION			(*Mode only for ReadCyclicPosition: use the value depending on the ctrl mode*)
	);

	MCEdgeEnum :
	(
		mcEDGE_POSITIVE,				(*change from logical low to logical high*)
		mcEDGE_NEGATIVE					(*change from logical high to logical low*)
	);

	MCBrakeCommandEnum :
	(
		mcBRAKE_CLOSE,					(*close brake*)
		mcBRAKE_OPEN,					(*open brake*)
		mcBRAKE_GET_STATUS				(*show status of brake*)
	);

	MCBrakeStatusEnum :
	(
		mcBRAKE_STATUS_NOT_PROVIDED,			(*command was not mcBRAKE_GET_STATUS*)
		mcBRAKE_CLOSED,					(*holding brake closed*)
		mcBRAKE_OPENED					(*holding brake open*)
	);

	MCSegmentProcessParIDModeEnum :
	(
		mcSEG_PARID_GET := 0, (*read ParID once from the segment*)
		mcSEG_PARID_SET	(*write ParID once to the segment*)
	);

	MCSegmentDataTypeEnum :
		(
		mcSEG_PARTYPE_BOOL := 1, (*data type BOOL*)
		mcSEG_PARTYPE_SINT, (*data type SINT*)
		mcSEG_PARTYPE_INT, (*data type INT*)
		mcSEG_PARTYPE_DINT, (*data type DINT*)
		mcSEG_PARTYPE_USINT, (*data type USINT*)
		mcSEG_PARTYPE_UINT, (*data type UINT*)
		mcSEG_PARTYPE_UDINT, (*data type UDINT*)
		mcSEG_PARTYPE_REAL, (*data type REAL*)
		mcSEG_PARTYPE_VOID := 65535  (*data type unknown*)
	);

	(*Structure types*)

	MCAdditionalGroupHome_15_Type : STRUCT
		HomingOrderSource : MCHomingOrderSourceEnum;	(*Source of the homing order*)
    	HomingOrder : ARRAY[0..14] OF UINT;				(*Specifies the homing order (see HomingOrder) The array is in ACS order.*)
	END_STRUCT;

	MCAdditionalStatusType : STRUCT
		TriggerSwitch1 : BOOL;
		TriggerSwitch2 : BOOL;
		DriveEnableSwitch : BOOL;
		ResetDone : BOOL;
		LagWarning : BOOL;
	END_STRUCT;

	MCAdvancedMoveCycParType : STRUCT
		Velocity : REAL;
		Acceleration : REAL;
		Deceleration : REAL;
		DisableJoltLimitation : BOOL;
	END_STRUCT;

	MCAdvancedVelCtrlParType : STRUCT
		Acceleration : REAL;
		Deceleration : REAL;
	END_STRUCT;

	MCAdvancedGearInParType : STRUCT
		MasterMaxVelocity : REAL;
	END_STRUCT;

	MCCamTableDefineType : STRUCT
		DataObjectName : STRING[12];
		DataAdress : UDINT;
	END_STRUCT;

	MCFrameOrientationType : STRUCT
		Type : UDINT;		(*Describes the representation of rotation angles 1 to 3*)
		Angle1 : LREAL;		(*Rotation angle 1 for describing the orientation*)
		Angle2 : LREAL;		(*Rotation angle 2 for describing the orientation*)
		Angle3 : LREAL;		(*Rotation angle 3 for describing the orientation*)
	END_STRUCT;

	MCFramePositionType : STRUCT
		X : LREAL;		(*Offset in the direction of the X-axis*)
		Y : LREAL;		(*Offset in the direction of the Y-axis*)
		Z : LREAL;		(*Offset in the direction of the Z-axis*)
	END_STRUCT;

	MCFrameType : STRUCT
		Trans : MCFramePositionType;	(*Position*)
		Rot : MCFrameOrientationType;	(*Orientation*)
	END_STRUCT;

	MCKinematicTrfType : UDINT;

	MCPrgInfoActiveProgramType : STRUCT 		(*Informations about the active program*)
		Name : STRING[260];						(*Name of the active program*)
		Number : UDINT;							(*Number of the active program*)
		Level : UINT;							(*Current program level*)
	END_STRUCT;

	MCPrgInfoBlockMonType : STRUCT (*Block monitor*)
		LineNumber : UDINT;				(*Current line number*)
		BlockNumber : UDINT;			(*Current block number*)
		LineLast2 : STRING[260];		(*Second to last line in the sequence program*)
		LineLast1 : STRING[260];		(*Last line in the sequence program*)
		LineActual : STRING[260];		(*Current line in the sequence program*)
		LineNext1 : STRING[260];		(*Next line in the sequence program*)
		LineNext2 : STRING[260];		(*Line following the next line in the sequence program*)
		RemainingDistance : LREAL;		(*Distance remaining until the end of the block [units]*)
		Length : LREAL;					(*Length of the path of the current block [units]*)
		LengthNext : LREAL;				(*Length of the path of the next block [units]*)
	END_STRUCT;

	MCPrgInfoPrgHierarchyLevelType : STRUCT  (*Program Hierarchy Levels*)
		LineNumber : UDINT;				(*Current level line number*)
	END_STRUCT;

	MCPrgInfoPrgHierarchyType : STRUCT (*Program Hierarchy*)
		Level : ARRAY[0..14] OF MCPrgInfoPrgHierarchyLevelType; (*Program Hierarchy Levels*)
	END_STRUCT;

	MCPrgInfoAxesMonType : STRUCT (*Axes Monitor*)
		Position : ARRAY[0..14] OF LREAL; (*Axes positions*)
	END_STRUCT;

	MCPrgInfoType : STRUCT (*The structure contains extended information about the running program*)
		InitProgram : STRING[260];						(*Name of the initialization subroutine*)
		ActiveProgram : MCPrgInfoActiveProgramType;		(*Information about the active program*)
		InterruptStatus : MCPrgInfoInterruptEnum;		(*Interrupt informations*)
		BlockMonitor : MCPrgInfoBlockMonType;			(*Block monitor*)
		ProgramHierarchy : MCPrgInfoPrgHierarchyType;	(*Program Hierarchy*)
	END_STRUCT;

	MCPrgInfo15Type : STRUCT (*The structure contains extended information about the running program*)
		InitProgram : STRING[260];						(*Name of the initialization subroutine*)
		ActiveProgram : MCPrgInfoActiveProgramType;		(*Information about the active program*)
		InterruptStatus : MCPrgInfoInterruptEnum;		(*Interrupt informations*)
		BlockMonitor : MCPrgInfoBlockMonType;			(*Block monitor*)
		ProgramHierarchy : MCPrgInfoPrgHierarchyType;	(*Program Hierarchy*)
		AxesMonitor : MCPrgInfoAxesMonType; 			(*Axes monitor*)
	END_STRUCT;

	MCPrgInfoParAxesMonType : STRUCT (*The structure contains parameters for the axes monitor*)
		CoordSystem : MCCoordinateSystemEnum; (*Define order of monitored axes*)
	END_STRUCT;

	MCPrgInfoParType : STRUCT (*The structure contains parameters for the program informations*)
		Mode : MCPrgInfoModeEnum; (*Source of monitored data*)
		AxesMonitor : MCPrgInfoParAxesMonType; (*The structure contains parameters for the axes monitor*)
	END_STRUCT;

	MCPrgAxesReposParType : STRUCT (*Axes repositioning parameters*)
		Type : MCPrgAxesReposTypeEnum;	(*Axes repositioning type*)
		String : STRING[260];			(*String Parameter*)
	END_STRUCT;

	MCPrgStartPointParRpcType : STRUCT (*Extended start point parameters for Rpc*)
		Level : UINT;									(*Program hierarchy level*)
		ProgramHierarchy : MCPrgInfoPrgHierarchyType;	(*Program Hierarchy*)
	END_STRUCT;

	MCTrackPathLimitsType : STRUCT (*Tracking path limit parameters*)
		Velocity : LREAL; 			(*Maximum path speed*)
		Acceleration : LREAL; 		(*Maximum path acceleration*)
		Deceleration : LREAL; 		(*Maximum path deceleration*)
		Jerk : LREAL; 				(*Maximum path jerk*)
	END_STRUCT;

	MCSegmentProcessParIDType : STRUCT
		ParID : UINT; (*ParID which is read/written*)
		VariableAddress : UDINT; (*address the value of the ParID is written to/read from*)
		DataType : MCSegmentDataTypeEnum; (*data type of the ParID value*)
	END_STRUCT;

	MCWorkspaceType : UDINT;	(*Function blocks with the input MCWorkspaceType receive a pointer to a STRING, which contains the name of the CNC program with the workspace definition.*)
	MCFFCtrlParType : UDINT;	(*Function blocks with the input MCFFCtrlParType receive a pointer to a parameter structure.*)
	MCPrgStartPointParExtType : UDINT; (*Function blocks with the input MCStartPointParExtType receive a pointer to a parameter structure.*)

	(*FB internals*)
	FubProcessing_csub : STRUCT (*Partial struct type (C only)*)
		states : ARRAY[0..1] OF DINT;
	END_STRUCT;

	TaskInteraction : FubProcessing_csub;

	MCInternalType : STRUCT (*internal variable*)
		ID : UDINT;
		Check : UDINT;
		ParamHash : UDINT;
		State : WORD;
		Error : UINT;
		Treating : REFERENCE TO TaskInteraction;
		Memory : ARRAY[0..13] OF UDINT;
		if_addr : UDINT;
	END_STRUCT;

	MCInternalTwoRefType : STRUCT (*internal variable*)
		ID : UDINT;
		Check : UDINT;
		ParamHash : UDINT;
		State : WORD;
		Error : UINT;
		Treating : REFERENCE TO TaskInteraction;
		Memory : ARRAY[0..13] OF UDINT;
		if_addr : UDINT;
		if_ma_addr : UDINT;
	END_STRUCT;

	IGmcAxisIf_csub : STRUCT (*Partial interface type (C only)*)
		vtable : DWORD;
	END_STRUCT;

	IGmcAxisIf : IGmcAxisIf_csub;

	GmcAxis : STRUCT
		controlif : REFERENCE TO IGmcAxisIf;
	END_STRUCT;

	IGmcAxesGrpIf_csub : STRUCT (*Partial interface type (C only)*)
		vtable : DWORD;
	END_STRUCT;
	IGmcAxesGrpIf : IGmcAxesGrpIf_csub;
	GmcAxesGroup : STRUCT
		controlif : REFERENCE TO IGmcAxesGrpIf;
	END_STRUCT;

	IGmcLLMIf_csub : STRUCT (*Partial interface type (C only)*)
		vtable : DWORD;
	END_STRUCT;
	IGmcLLMIf : IGmcLLMIf_csub;
	GmcLLMAssembly : STRUCT
		controlif : REFERENCE TO IGmcLLMIf;
	END_STRUCT;

	IGmcLLMSegIf_csub : STRUCT (*Partial interface type (C only)*)
		vtable : DWORD;
	END_STRUCT;
	IGmcLLMSegIf : IGmcLLMSegIf_csub;
	GmcLLMSegment : STRUCT
		controlif : REFERENCE TO IGmcLLMSegIf;
	END_STRUCT;

	IGmcLLMSectorIf_csub : STRUCT (*Partial interface type (C only)*)
		vtable : DWORD;
	END_STRUCT;
	IGmcLLMSectorIf : IGmcLLMSectorIf_csub;
	GmcLLMSector : STRUCT
		controlif : REFERENCE TO IGmcLLMSectorIf;
	END_STRUCT;

END_TYPE
```

### MAPPSuppor.var
```iecst
(********************************************************************
 * COPYRIGHT -- Microsoft
 ********************************************************************
 * Library: MAPPSuppor
 * File: MAPPSuppor.var
 * Author: John
 * Created: April 23, 2015
 ********************************************************************
 * Constants of library MAPPSuppor
 ********************************************************************)
VAR CONSTANT
	DEFINE_LOGSTRING_LEN : UDINT := 512;
	MAX_CALLS_INIT_LOGBOOK : UDINT := 50;
	MAX_IDX_LANGUAGES : UDINT := 5;
	DEFINE_LANGUAGE_STRINGS : ARRAY[0..MAX_IDX_LANGUAGES] OF STRING[4] := ['en','sv','pt','de','es','fr']; (*MUST MATCH EXACTLY THE LANGUAGES IN THE ORDER THEY ARE CONFIGURED IN PROJECT LANGUAGES.*)
	DEFINE_MAX_IDX_HMI_TABLES : UDINT := 3;
	DEFINE_MAX_TABLE_ENTRIES : UDINT := 20;
	DEFINE_PAR_DESC_MAXLEN : UDINT := 240;
	DEFINE_PAR_NAME_MAXLEN : UDINT := 80;
	DEFINE_PAR_IDX_MAXLEN : UDINT := 4;
END_VAR
(*Insert your comment here.*)
VAR CONSTANT
	Enum_Max_Listbox_Char : USINT := 80;
	Enum_Max_Listbox_Items : USINT := 12;
END_VAR
(*Insert your comment here.*)
VAR CONSTANT
	HMI_ENUM_TAB_KEYS_MAX : USINT := 11;
	HMI_ENUM_MENU_ITEMS_RT : USINT := 11;
	HMI_ENUM_MENU_ITEMS_LT : USINT := 11;
END_VAR
(*Insert your comment here.*)
VAR CONSTANT
	HMI_PWD_MAXLEN : UDINT := 15;
	HMI_PWD_LEVELS : UDINT := 4;
END_VAR
(*Insert your comment here.*)
VAR CONSTANT
	DEFINE_INDEX_TEXTTABLE_PV : USINT := LANGUAGE_ENGLISH;
	DEFINE_INDEX_TEXTTABLE_DEFAULT : USINT := LANGUAGE_SWEDISH;
	DEFINE_INDEX_TEXTTABLE_MIN : USINT := LANGUAGE_PORTUGESE;
	DEFINE_INDEX_TEXTTABLE_MAX : USINT := LANGUAGE_GERMAN;
	DEFINE_INDEX_TEXTTABLE_HIDE : USINT := LANGUAGE_SPANISH;
END_VAR
```

### MTFilter.var
```iecst
(*Error*)
VAR CONSTANT
	mtBCD_ERR_FILTER_TYPE_INVALID : DINT := -1058012158; (*Filter type is invalid.*)
	mtBCD_ERR_FILTER_ORDER_INVALID : DINT := -1058012157; (*Filter order is invalid.*)
	mtBCD_ERR_CUTOFF_FREQ_INVALID : DINT := -1058012156; (*Cutoff frequency of the filter is invalid.*)
	mtBCD_ERR_CENTER_FREQ_INVALID : DINT := -1058012155; (*Center frequency of the filter is invalid.*)
	mtBCD_ERR_FILTER_BANDWIDTH : DINT := -1058012154; (*Bandwidth of the filter is invalid.*)
	mtBCD_ERR_FREQ_NUM_INVALID : DINT := -1058012153; (*Filter frequency of the numerator is invalid.*)
	mtBCD_ERR_DAMPING_NUM_INVALID : DINT := -1058012152; (*Damping of the numerator is invalid.*)
	mtBCD_ERR_FREQ_DEN_INVALID : DINT := -1058012151; (*Filter frequency of the denominator is invalid.*)
	mtBCD_ERR_DAMPING_DEN_INVALID : DINT := -1058012150; (*Damping of the denominator is invalid.*)
	mtBCD_ERR_FILTER_WINDOW_INVALID : DINT := -1058012149; (*Window length of the filter is invalid.*)
END_VAR
(*Warning*)
VAR CONSTANT
	mtBCD_WRN_FILTER_TYPE_INVALID : DINT := -2131753982; (*Filter type is invalid.*)
	mtBCD_WRN_FILTER_ORDER_INVALID : DINT := -2131753981; (*Filter order is invalid.*)
	mtBCD_WRN_CUTOFF_FREQ_INVALID : DINT := -2131753980; (*Cutoff frequency of the filter is invalid.*)
	mtBCD_WRN_CENTER_FREQ_INVALID : DINT := -2131753979; (*Center frequency of the filter is invalid.*)
	mtBCD_WRN_FILTER_BANDWIDTH : DINT := -2131753978; (*Bandwidth of the filter is invalid. *)
	mtBCD_WRN_FREQ_NUM_INVALID : DINT := -2131753977; (*Filter frequency of the numerator is invalid. *)
	mtBCD_WRN_DAMPING_NUM_INVALID : DINT := -2131753976; (*Damping of the numerator is invalid. *)
	mtBCD_WRN_FREQ_DEN_INVALID : DINT := -2131753975; (*Filter frequency of the denominator is invalid. *)
	mtBCD_WRN_DAMPING_DEN_INVALID : DINT := -2131753974; (*Damping of the denominator is invalid. *)
	mtBCD_WRN_FILTER_WINDOW_INVALID : DINT := -2131753973; (*Window length of the filter is invalid. *)
END_VAR
```

### MTProfile.typ
```iecst
TYPE
	MTProfileFunctionModeEnum :
		( (*Interpolation modes.*)
		mtPROFILE_ZERO_ORDER_HOLD := 0, (*Zero-Order-Hold (incremental) interpolation.*)
		mtPROFILE_FIRST_ORDER_HOLD := 1 (*First-Order-Hold (linear) interpolation.*)
		);
	MTProfilePositionStateEnum :
		(
		mtPROFILE_DEC_NEG_DIR := -3, (*Deceleration phase, negative direction of movement.*)
		mtPROFILE_CONST_VEL_NEG_DIR := -2, (*Constant velocity phase, negative direction of movement.*)
		mtPROFILE_ACC_NEG_DIR := -1, (*Acceleration phase, negative direction of movement.*)
		mtPROFILE_STANDSTILL := 0, (*Standstill.*)
		mtPROFILE_ACC_POS_DIR := 1, (*Acceleration phase, positive direction of movement.*)
		mtPROFILE_CONST_VEL_POS_DIR := 2, (*Constant velocity phase, positive direction of movement.*)
		mtPROFILE_DEC_POS_DIR := 3 (*Deceleration phase, positive direction of movement.*)
		);
	MTProfilePositionParameterType : 	STRUCT  (*Movement parameters.*)
		VelocityPosDirection : REAL; (*Maximum velocity of movement in the "positive" direction. Unit: [Units/s]. Valid value range: VelocityPosDirection > 0.*)
		VelocityNegDirection : REAL; (*Maximum velocity of movement in the "negative" direction. Unit: [Units/s]. Valid value range: VelocityNegDirection > 0.*)
		AccelerationPosDirection : REAL; (*Maximum acceleration when moving in the "positive" direction. Unit: [Units/s�]. Valid value range: AccelerationPosDirection > 0.*)
		DecelerationPosDirection : REAL; (*Maximum deceleration when moving in the "positive" direction. Unit: [Units/s�]. Valid value range: DecelerationPosDirection > 0.*)
		AccelerationNegDirection : REAL; (*Maximum acceleration when moving in the "negative" direction. Unit: [Units/s�]. Valid value range: AccelerationNegDirection > 0.*)
		DecelerationNegDirection : REAL; (*Maximum deceleration when moving in the "negative" direction. Unit: [Units/s�]. Valid value range: DecelerationNegDirection > 0.*)
		JoltTime : REAL; (*Jolt limit time. Unit: [s]. Valid value range: 0 <= JoltTime <= "10000 � task cycle time".*)
	END_STRUCT;
	MTProfileFunctionNodeType : 	STRUCT  (*Interpolation point.*)
		TimeValue : REAL; (*Time coordinate of an interpolation point in the array. Unit: [s]. Valid value range: TimeValue >= 0.*)
		FcnValue : REAL; (*Function value of an interpolation point in the array.*)
		Internal : MTProfileFcnNodeInternalType; (*Data for internal use.*)
	END_STRUCT;
	MTProfileFcnNodeInternalType : 	STRUCT  (*Internal variables of an interpolation point.*)
		TimeValue : REAL; (*Data for internal use.*)
		FcnValue : REAL; (*Data for internal use.*)
		C0 : REAL; (*Data for internal use.*)
		C1 : REAL; (*Data for internal use.*)
	END_STRUCT;
	MTProfilePosGenInternalType : 	STRUCT  (*Internal variables of function block MTProfilePositionGenerator.*)
		CycleTime : REAL; (*Task cycle time. Unit: [탎].*)
		Tv : ARRAY[0..2]OF LREAL; (*Data for internal use.*)
		ParametersValid : BOOL; (*Data for internal use.*)
		Parameter : MTProfilePositionParameterType; (*Data for internal use.*)
		ProfileNb : USINT; (*Data for internal use.*)
		ProfileID : USINT; (*Data for internal use.*)
		MovementCase : SINT; (*Data for internal use.*)
		MovementPhase : USINT; (*Data for internal use.*)
		MovementStep : USINT; (*Data for internal use.*)
		HomeVelocity : REAL; (*Data for internal use.*)
		HomeVelocityIntrude : USINT; (*Data for internal use.*)
		HomeVelocityDbl : LREAL; (*Data for internal use.*)
		HomeVelocityState : USINT; (*Data for internal use.*)
		Quantum0 : LREAL; (*Data for internal use.*)
		Quantum : REAL; (*Data for internal use.*)
		QuantumJolt : REAL; (*Data for internal use.*)
		QuantumSPF : LREAL; (*Data for internal use.*)
		Position0 : LREAL; (*Data for internal use.*)
		Position : REAL; (*Data for internal use.*)
		PositionJolt : REAL; (*Data for internal use.*)
		PositionSPF : LREAL; (*Data for internal use.*)
		PositionOffset : LREAL; (*Data for internal use.*)
		Velocity0 : LREAL; (*Data for internal use.*)
		Velocity : REAL; (*Data for internal use.*)
		VelocityJolt : REAL; (*Data for internal use.*)
		VelocitySPF : LREAL; (*Data for internal use.*)
		Acceleration0 : LREAL; (*Data for internal use.*)
		Acceleration : REAL; (*Data for internal use.*)
		AccelerationJolt : REAL; (*Data for internal use.*)
		AccelerationSPF : LREAL; (*Data for internal use.*)
		JoltTimeMax : REAL; (*Data for internal use.*)
		JoltTime : LREAL; (*Data for internal use.*)
		EndPosition : REAL; (*Data for internal use.*)
		PositionDifference : LREAL; (*Data for internal use.*)
		BrakingDistance : LREAL; (*Data for internal use.*)
		TopSpeed : LREAL; (*Data for internal use.*)
		ParameterV : ARRAY[0..5]OF REAL; (*Data for internal use.*)
		AccelerationV : ARRAY[0..19]OF LREAL; (*Data for internal use.*)
		ConstantV : ARRAY[0..19]OF LREAL; (*Data for internal use.*)
		DecelerationV : ARRAY[0..19]OF LREAL; (*Data for internal use.*)
		TimerV : ARRAY[0..1]OF LREAL; (*Data for internal use.*)
		QuantumBuffer : REFERENCE TO LREAL; (*Data for internal use.*)
		PositionBuffer : REFERENCE TO LREAL; (*Data for internal use.*)
		VelocityBuffer : REFERENCE TO LREAL; (*Data for internal use.*)
		AccelerationBuffer : REFERENCE TO LREAL; (*Data for internal use.*)
		BufCntMax : DINT; (*Data for internal use.*)
		BufCnt : DINT; (*Data for internal use.*)
		CntJoltTime : DINT; (*Data for internal use.*)
		BufCntJoltTime : DINT; (*Data for internal use.*)
		AtStandstill : BOOL; (*Data for internal use.*)
		ExecutionEvent : USINT; (*Data for internal use.*)
		Start : BOOL; (*Data for internal use.*)
		StartOld : BOOL; (*Data for internal use.*)
		Stop : BOOL; (*Data for internal use.*)
		StopOld : BOOL; (*Data for internal use.*)
		AbortOld : BOOL; (*Data for internal use.*)
		SetHomePositionOld : BOOL; (*Data for internal use.*)
		Update : BOOL; (*Data for internal use.*)
		UpdateOld : BOOL; (*Data for internal use.*)
		EnableOld : BOOL; (*Data for internal use.*)
		SystemInfo : SysInfo; (*Internally used function block.*)
		ConstTaskCycle : BOOL; (*Data for internal use.*)
		TimeCounterState : UINT; (*Data for internal use.*)
		MicroSecondsOld : UDINT; (*Data for internal use.*)
		SystemTicksOld : UDINT; (*Data for internal use.*)
		MemStatus : UINT;
		BufLen : UDINT;
		TCycle : REAL; (*TCycle = 0 for the first run and TCycle=Ts for all the others.*)
	END_STRUCT;
	MTProfileFcnGenInternalType : 	STRUCT  (*Internal variables of function block MTProfileFcnGenerator.*)
		CycleTime : REAL; (*Task cycle time. Unit: [탎].*)
		Tv : ARRAY[0..1]OF LREAL; (*Data for internal use.*)
		ParametersValid : BOOL; (*Data for internal use.*)
		Nodes : REFERENCE TO MTProfileFunctionNodeType; (*Data for internal use.*)
		NumberOfNodes : UINT; (*Data for internal use.*)
		TimeValueOrder : SINT; (*Data for internal use.*)
		Period : REAL; (*Data for internal use.*)
		TimerV : ARRAY[0..1]OF LREAL; (*Data for internal use.*)
		ResetTimer : BOOL; (*Data for internal use.*)
		Update : BOOL; (*Data for internal use.*)
		UpdateOld : BOOL; (*Data for internal use.*)
		EnableOld : BOOL; (*Data for internal use.*)
		Bootkey : UDINT; (*Data for internal use.*)
		SystemInfo : SysInfo; (*Internally used function block.*)
		ConstTaskCycle : BOOL; (*Data for internal use.*)
		TimeCounterState : UINT; (*Data for internal use.*)
		MicroSecondsOld : UDINT; (*Data for internal use.*)
		SystemTicksOld : UDINT; (*Data for internal use.*)
		BootkeyTimeCounter : UDINT; (*Data for internal use.*)
		PerTemp : REAL; (*Temporary period*)
		TCycle : REAL; (*TCycle = 0 for the first run and TCycle=Ts for all the others.*)
	END_STRUCT;
END_TYPE
```

### Visapi.var
```iecst
(********************************************************************
 * COPYRIGHT -- Bernecker + Rainer
 ********************************************************************
 * Library: Visapi
 * File: Visapi.var
 * Created: 11.11.2003
 ********************************************************************
 *
 ********************************************************************)
VAR CONSTANT
	vaERR_VISAPI_NOT_INITIALIZED : UINT := 100; (*visapi not initialized*)
	vaERR_RESOURCE_WRONG_FORMAT : UINT := 7197; (*resource has wrong format*)
	vaERR_RESOURCE_NOT_FOUND : UINT := 7196; (*resource not found*)
	vaERR_NO_MORE : UINT := 7195; (*no data found*)
	vaERR_ALREADY : UINT := 7190; (*connection already exists*)
	vaERR_RESOURCES : UINT := 7180; (*resource error*)
	vaERR_MEMORY : UINT := 7170; (*no memory*)
	vaERR_VERSION : UINT := 7160; (*version conflict*)
	vaERR_ARGUMENT : UINT := 7150; (*wrong arguments*)
	vaERR_TIMEOUT : UINT := 7140; (*timeout*)
	vaERR_CONNECTION_LOST : UINT := 7130; (*connection lost*)
	vaERR_OVERFLOW : UINT := 7120; (*memory overflow*)
	vaERR_ACCESS : UINT := 7111; (*access error*)
	vaERR_NO_ACCESS : UINT := 7110; (*access error*)
	vaERR_EXISTS : UINT := 7101; (*resource exists already*)
	vaERR_CREATE_TASK_FAILED : UINT := 7100; (*create task failed*)
	vaERR_PARAMETER : UINT := 7090; (*parameter error*)
	vaERR_NOT_SUPPORTED : UINT := 7080; (*function not supported*)
	vaERR_KEYMATRIX_NOT_VALID : UINT := 7070; (*keymatrix not valid*)
	vaERR_FONTMODULE_NOT_FOUND : UINT := 7060; (*fontmodul no found*)
	vaERR_UNDEFINED_ERROR_CODE : UINT := 7050; (*undefined error code*)
	vaERR_WRONG_MODULE_NAME : UINT := 7030; (*wrong module name*)
	vaERR_DRIVER_NOT_FOUND : UINT := 7020; (*driver not found*)
	vaERR_INTERPRETER_NOT_READY : UINT := 7010; (*interpreter not ready*)
	vaERR_BUSY_ALARMSYSTEM : UINT := 247; (*alarmsystem busy*)
	vaERR_DELHISLIST : UINT := 246; (*error delting alarm history*)
	vaERR_NOALARMQUIT : UINT := 245; (*error in quiting alarm*)
	vaERR_EMPTY_ALARMLIST : UINT := 240; (*empty alarm list*)
	vaERR_BUSY : UINT := 7000; (*busy*)
	vaERR_EMPTY_HISTORYLIST : UINT := 248; (*empty alarm history*)

	vaALS_INACTIVE :UDINT := 1; (*Filter for inactive alarms*)
 	vaALS_ACTIVE :UDINT := 2; (*Filter for active alarms*)
	vaALS_ACKNOWLEDGED :UDINT := 16; (*Filter for acknowledged alarms*)
	vaALS_NOTACKNOWLEDGED :UDINT := 32; (*Filter for not acknowledged alarms*)
	vaALS_BYPASSSED :UDINT := 256; (*Filter for bypassed alarms*)
	vaALS_NOTBYPASSSED :UDINT := 512; (*Filter for not bypassed alarms*)
 	vaALS_CURRENT :UDINT := 16#10000; (*Filter for current alarms*)
END_VAR
```

### Package Logical/UserLibraries/wbrServices - Service libraries

### Library Logical/UserLibraries/wbrServices/bglibasWBR (ANSIC)
Depends on: standard, wbrLogSvc

### Program Logical/UserLibraries/wbrServices/Cyclic/wbrService (ANSIC)

#### wbrServiceCyclic.c - Cyclic code
```c
/*!
 ********************************************************************
### Program : wbrService
 * \file :   wbrServiceCyclic.c
 * \author : Blanton Radford
 * \date Created: May 18, 2015
 * \copyright -- Piedmont Automation
 ********************************************************************
 * \brief Cyclic updates for the package WBRServices
 ********************************************************************/

#ifdef _DEFAULT_INCLUDES
  #include <AsDefault.h>
#endif

/*! \brief Cyclic task for WBRServices
*   \pre   Place in TC#8 after most if not all other tasks
*/
void _CYCLIC wbrServiceCyclic(void)
{
  //! \todo   check available mem and set flags to increase partition size if needed
  memService.status.blockFree=  memSvcGetMemInfo(&memService);

  if(logService.busy)  writeMessagesToLog();

  wbrPingStation(&genericPing);

  wbrUSBMonitor();
}

void _EXIT wbrServiceExit(void)
{
  if(logService.busy)  writeMessagesToLog();
}
```

#### wbrUSBService.c
```c
/*!
 ********************************************************************
### Program : wbrService
 * \file :   wbrUSBService.c
 * \author : Blanton Radford
 * \date Created: November 02, 2016
 * \copyright -- Piedmont Automation
 ********************************************************************
 * \brief Cyclic updates for the package WBRServices
 ********************************************************************/

#ifdef _DEFAULT_INCLUDES
  #include <AsDefault.h>
#endif

#include  <string.h>

// int   usb->nextNodeIdx=  0;
// _LOCAL  USINT stringDescriptorIndex;

/*————————————————————————————————————————————————————————————————————————————*/
/*! \brief Monitor USB device ready, destroy if false
    \pre

rtyp              ƒ(x)————————¬  —argument comments—————————————————————————•••™  */

static  void  monitorNodeReady(

        wbrUSBService_typ * usb                     //!<
      )
{
 int  i;

  for(i=0;  i < wbrusbNUM_NODES;  i++)  {
    if(   usb->node[i].deviceData.interfaceClass == asusb_CLASS_MASS_STORAGE
       && usb->node[i].isActive == 1)
    {

      UsbMsDeviceReady(&usb->node[i].fbMonStorageReady);

      if(usb->node[i].fbMonStorageReady.status == wbrSvc_AsFBStatus_SUCCESS ) {
        usb->node[i].isReady= 1;
        usbServiceIF[i].isReady= 1;
        usbServiceIF[i].isFileIODevice= 1;
        continue;
      }
      if(usb->node[i].fbMonStorageReady.status == asusbERR_USB_NOTFOUND)   {
        memset( &usb->node[i]
              , 0
              , sizeof(usb->node[i]) - sizeof(usb->node[i].fbMonStorageReady)
              );
        memset( &usbServiceIF[i]
              , 0
              , sizeof(usbServiceIF[i])
              );
        if( i < usb->nextNodeIdx )    usb->nextNodeIdx= i;
      }
    }
  }
}
/*————————————————————————————————————————————————————————————————————————————*/

/*————————————————————————————————————————————————————————————————————————————*/
/*! \brief Monitor for changes in the USB node list from FB
    \pre

rtyp              ƒ(x)————————¬  —argument comments—————————————————————————•••™  */

static  BOOL  monitorChangesInNodeList(

        wbrUSBService_typ * usb                     //!<
      )
{
 int  i, j;

 BOOL
        idExists= 0;
      ;

  usb->list.fb.enable = 1;
  usb->list.fb.pBuffer = (UDINT)&usb->list.listCurr;
  usb->list.fb.bufferSize = sizeof(usb->list.listCurr);
  usb->list.fb.filterInterfaceClass = 0;
  usb->list.fb.filterInterfaceSubClass = 0;
  UsbNodeListGet(&usb->list.fb);

  switch(usb->list.fb.status)    {
   case 32900:   // case asusbERR_USB_NOTFOUND:
    monitorNodeReady(usb);
    return  0;

   case wbrSvc_AsFBStatus_SUCCESS:
    for(i=0;  i < wbrusbNUM_NODES;  i++)  {
      if(usb->list.listCurr[i] != usb->list.listPrev[i])  {
        for(j=0;  j < wbrusbNUM_NODES; j++)
          if(usb->list.listCurr[i] == usb->list.listPrev[j])  {

            idExists= 1;
            break;    //  nodeID already in list
          }
        if(idExists)  {
          idExists= 0;
          usb->list.listPrev[i]=  usb->list.listCurr[i];
          continue;
        }
        usb->list.listPrev[i]=  usb->list.listCurr[i];
        usb->list.newNodeDetected=  1;

        usb->node[usb->nextNodeIdx].string[0].isWorking=
              usb->node[usb->nextNodeIdx].string[1].isWorking=
              usb->node[usb->nextNodeIdx].string[2].isWorking=
              usb->node[usb->nextNodeIdx].string[3].isWorking=
            usb->node[usb->nextNodeIdx].isWorking= 1;

        usb->node[usb->nextNodeIdx].fbGetNode.nodeId=
              usb->node[usb->nextNodeIdx].fbGetDescDev.nodeId=
              usb->node[usb->nextNodeIdx].string[0].fb.nodeId=
              usb->node[usb->nextNodeIdx].string[1].fb.nodeId=
              usb->node[usb->nextNodeIdx].string[2].fb.nodeId=
              usb->node[usb->nextNodeIdx].string[3].fb.nodeId=
            usb->list.listCurr[i];
        usb->node[usb->nextNodeIdx].isNew= 1;

        usb->node[usb->nextNodeIdx].fbGetNode.enable=      1;
        usb->node[usb->nextNodeIdx].fbGetNode.pBuffer=
            (UDINT)&usb->node[usb->nextNodeIdx].deviceData;
        usb->node[usb->nextNodeIdx].fbGetNode.bufferSize=
            sizeof(usb->node[usb->nextNodeIdx].deviceData);

        UsbNodeGet(&usb->node[usb->nextNodeIdx].fbGetNode);

        usb->node[usb->nextNodeIdx].string[0].fb.enable=
            usb->node[usb->nextNodeIdx].fbGetDescDev.enable=      1;
        usb->node[usb->nextNodeIdx].fbGetDescDev.requestType=     asusb_USB_RT_DEVICE;
        usb->node[usb->nextNodeIdx].fbGetDescDev.descriptorType=  asusb_USB_DESCR_DEVICE;
        usb->node[usb->nextNodeIdx].string[0].fb.requestType=     asusb_USB_RT_DEVICE;
        usb->node[usb->nextNodeIdx].string[0].fb.descriptorType=  asusb_USB_DESCR_STRING;
        usb->node[usb->nextNodeIdx].string[0].fb.descriptorIndex=
            usb->node[usb->nextNodeIdx].fbGetDescDev.descriptorIndex= 0;
        usb->node[usb->nextNodeIdx].string[0].fb.languageId=
            usb->node[usb->nextNodeIdx].fbGetDescDev.languageId=      0;
        usb->node[usb->nextNodeIdx].fbGetDescDev.pBuffer=
            (UDINT)&usb->node[usb->nextNodeIdx].deviceDescriptor;
        usb->node[usb->nextNodeIdx].fbGetDescDev.bufferSize=
            sizeof(usb->node[usb->nextNodeIdx].deviceDescriptor);
        usb->node[usb->nextNodeIdx].string[0].fb.pBuffer=
            (UDINT)&usb->node[usb->nextNodeIdx].string[0].descriptor;
        usb->node[usb->nextNodeIdx].string[0].fb.bufferSize=
              sizeof(usb->node[usb->nextNodeIdx].string[0].descriptor)
            + sizeof(usb->node[usb->nextNodeIdx].string[0].descContainer);

        UsbDescriptorGet(&usb->node[usb->nextNodeIdx].fbGetDescDev);
        UsbDescriptorGet(&usb->node[usb->nextNodeIdx].string[0].fb);

        //  find next empty node
        usb->nextNodeIdx++;
        for(  ; usb->node[usb->nextNodeIdx].isActive; usb->nextNodeIdx++) {}

      }
    }
    break;

   case 32901:   // case asusbERR_BUFSIZE:
   case 32902:   // case asusbERR_NULLPOINTER:
    /* Error Handling */
   default:
    break;
  }

  return  (BOOL)usb->list.fb.listNodes;
}
/*————————————————————————————————————————————————————————————————————————————*/

/*————————————————————————————————————————————————————————————————————————————*/
/*! \brief Get node data using FBs, publish device name
    \pre

rtyp              ƒ(x)————————¬  —argument comments—————————————————————————•••™  */

static  void  getNodeDataAndPublishDeviceLinkInfo(

        wbrUSBService_typ * usb                     //!<
      )
{
 int  i, j;

  usb->list.newNodeDetected=  0;

  for(i=0;  i < wbrusbNUM_NODES;  i++)  {
    /// \todo  if node empty && usb->nextNodeIdx > i, usb->nextNodeIdx=  i;
    if(usb->node[i].isNew == 0)   continue;

    switch(usb->node[i].fbGetNode.status)      {
     case wbrSvc_AsFBStatus_BUSY:

      UsbNodeGet(&usb->node[i].fbGetNode);

      if(usb->node[i].fbGetNode.status  == wbrSvc_AsFBStatus_BUSY)
        break;

     case wbrSvc_AsFBStatus_SUCCESS:
      usb->node[i].isActive=  1;

      if(usb->node[i].deviceData.interfaceClass == asusb_CLASS_MASS_STORAGE) {
        wbrsnprintf(usbServiceIF[i].fileIODeviceParam
                  , sizeof(usbServiceIF[i].fileIODeviceParam)
                  , "/DEVICE=%s"
                  , usb->node[i].deviceData.ifName
                  );
        usb->node[i].fbMonStorageReady.enable=  1;
        usb->node[i].fbMonStorageReady.pIfName= (UDINT)usb->node[i].deviceData.ifName;
      }
      usb->node[i].fbGetNode.status++;
      break;

     case 32900:   // case asusbERR_USB_NOTFOUND:
     case 32901:   // case asusbERR_BUFSIZE:
     case 32902:   // case asusbERR_NULLPOINTER:
      break;
    }

    switch(usb->node[i].fbGetDescDev.status)      {
     case wbrSvc_AsFBStatus_BUSY:

      UsbDescriptorGet(&usb->node[i].fbGetDescDev);

      if(usb->node[i].fbGetDescDev.status  == wbrSvc_AsFBStatus_BUSY)
        break;

     case wbrSvc_AsFBStatus_SUCCESS:
      usb->node[i].string[1].fb.descriptorIndex=
          usb->node[i].deviceDescriptor.manufacturerIndex;
      usb->node[i].string[2].fb.descriptorIndex=
          usb->node[i].deviceDescriptor.productIndex;
      usb->node[i].string[3].fb.descriptorIndex=
          usb->node[i].deviceDescriptor.serialNumberIndex;

      for(j=1;  j < 4;  j++)  {
        usb->node[i].string[j].fb.enable=          1;
        usb->node[i].string[j].fb.requestType=     asusb_USB_RT_DEVICE;
        usb->node[i].string[j].fb.descriptorType=  asusb_USB_DESCR_STRING;
        usb->node[i].string[j].fb.languageId=      0;
        usb->node[i].string[j].fb.pBuffer=
            (UDINT)&usb->node[i].string[j].descriptor;
        usb->node[i].string[j].fb.bufferSize=
              sizeof(usb->node[i].string[j].descriptor)
            + sizeof(usb->node[i].string[j].descContainer);

        UsbDescriptorGet(&usb->node[i].string[j].fb);
      }
      usb->node[i].isWorking= 0;
      usb->node[i].fbGetDescDev.status++;
      break;

     case 32900:   // case asusbERR_USB_NOTFOUND:
     case 32901:   // case asusbERR_BUFSIZE:
     case 32902:   // case asusbERR_NULLPOINTER:
      break;
    }

    for(j=0;  j < 4;  j++)  {
      switch(usb->node[i].string[j].fb.status)      {
       case wbrSvc_AsFBStatus_BUSY:

          UsbDescriptorGet(&usb->node[i].string[j].fb);

        if(usb->node[i].string[j].fb.status  == wbrSvc_AsFBStatus_BUSY)
          break;

       case wbrSvc_AsFBStatus_SUCCESS:
        usb->node[i].string[j].isWorking= 0;
        break;

       case 32900:   // case asusbERR_USB_NOTFOUND:
       case 32901:   // case asusbERR_BUFSIZE:
       case 32902:   // case asusbERR_NULLPOINTER:
        break;
      }
    }

    if(   usb->node[i].isWorking            == NO
       && usb->node[i].string[0].isWorking  == NO
       && usb->node[i].string[1].isWorking  == NO
       && usb->node[i].string[2].isWorking  == NO
       && usb->node[i].string[3].isWorking  == NO)
    {
      usb->node[i].isNew= 0;
    }
    else  {
      usb->list.newNodeDetected=  1;
    }
  }
}
/*————————————————————————————————————————————————————————————————————————————*/

/*————————————————————————————————————————————————————————————————————————————*/
/*! \brief Monitor USB device ready, destroy if false
    \pre

rtyp              ƒ(x)————————¬  —argument comments—————————————————————————•••™  */

void  wbrUSBMonitor(

        // usbNode_typ usbNode                     //!<
      )
{
  if(!monitorChangesInNodeList(&usbService))   return;

  if(usbService.list.newNodeDetected)  {
    // for(i=0; i< ; i++){
      getNodeDataAndPublishDeviceLinkInfo(&usbService);

    // }
  }

  monitorNodeReady(&usbService);
}
/*————————————————————————————————————————————————————————————————————————————*/
```

### changeLog.txt
```
TODO:
!!! clean up listSvc mem usage!!!
                              - add code to trim e.g. 10% from log lists when mem usage reaches a certain point
                              x - move mem mgt to new lib wbrMemSvc
                              - add code to increase heap block request if usage > e.g. 50%
                              - add code to warn when heap block usage > e.g. 90%

LogSvc                        x - don't use list if status == 0 after first func call
                              x - get rid of fb pointer if possible - keeping but handled better
                              - implement logging level
                              - link multiple messages/events together using Origin
                              - individual logs for libraries
                                - support for upstream services, e.g. listSvc

wbrIOSvc
wbrNetSvc
wbrStrUtil

wbrsprintf                    - try preprocessor trick in header to allow dynamic lib
                                - #ifdef prototypes to prevent use in static lib
                                - add static lib as dependency of dynamic lib
                                - define the token used in #ifdef in dynamic lib so that prototypes are linked there

0.11.0  2016-09
  Imported TimerServices updates from Hailo GLOBALlift/TOPlift
  ListSvc
    CharListToStringArray
      Add maxNodes to control log size - Fixed mem leak!
      Print element numbers with text
      Some cleanup
    Some cleanup
  LogSvc
    text logs
      separate printing and display updates
      more control using existing and new ListSvc features
      updated Init
    Fixed possible crash when declaring fb if mem alloc during node declaration fails, i.e. node == 0
    Begin conversion to ArEventLog from AsArLog
      Convert logbook get ident - it appears other info is no longer necessary
      Convert logbook creation
    Some cleanup
  PingSvc
    improved logging
      fixed logbook entry failure
      added fb not enabled as error msg
      less logbook spamming on ping success, and more control over the logging of success
      fixed errors when changing target station
    \todo   move wbrSQL_DT2_ISOFmtdStringFromDT() to wbrStrUtil
  Removed unused packages
  runFirstInit
    added asConfigID
    added version to compile info completed msg

0.10.8  2016-05-03
  Published to J. Glisson.  Used without issues as of 2016-09-13

0.10.7  2016-04
  Clean up some /todos and other comments
  Added wbrMemService to wrap AsMem and allow services besides list service
    to use heap memory
    moved mem funcs and data from wbrListService to wbrMemService

0.10.6  2016-03-31
  Added TimerServices
    Made a few mods to suit Hailo project and be more generic, e.g. msTimer object declared
    Using clock_ms() from AsTime to count milliseconds
    Added msTimer.diff_ms to facilitate time tracking, e.g. "hour meters"
  A few changes to Init and Cyclic to be more generic for multiple projects
    Write compile info to log on Init
  Updated package dependencies to facilitate more trouble-free importing

0.10.5  2015-10-??
  Initial release
    Used in APDW project
    No complaints as of 2016-03-07
```

### appConfig.typ
```iecst
(********************************************************************
 * COPYRIGHT --
 ********************************************************************
 * Package: ConfigAndRecipes
 * File: appConfig.typ
 * Author: goran_2
 * Created: August 06, 2011
 ********************************************************************
 * Data types of package ConfigAndRecipes
 ********************************************************************)
(*Insert your comment here.*)

TYPE
	cfgMachineConfig_typ : 	STRUCT  (*Machine configuration includes settings for timers and settings for servo drives.*)
		cfgFile : cfgFileInfo_typ;
		cfgCompile : cfgCompileVersionInfo_typ;
		wbrMemService : wbrMemSvcStoredConfig_typ;
	END_STRUCT;
END_TYPE
```

- Program Logical/UserLibraries/wbrServices/InitSP/runFirst (ANSIC) (no source held here)

### Library Logical/UserLibraries/wbrServices/wbrListSvc (ANSIC)
Depends on: wbrsprintf, wbrMemSvc

#### wbrListSvc.fun - Exported functions and function blocks
```iecst
(********************************************************************
 * COPYRIGHT -- Piedmont Automation
 ********************************************************************
 * Library: wbrListSvc
 * File: wbrListSvc.fun
 * Author: Blanton Radford
 * Created: May 07, 2015
 ********************************************************************
 * Functions and function blocks of library wbrListSvc
 ********************************************************************)

FUNCTION listSvcRequestListNode : UDINT
	VAR_INPUT
		l : linkedList_typ;
	END_VAR
END_FUNCTION

FUNCTION listSvcRequestList : UDINT
	VAR_INPUT
		size : UDINT;
		kind : linkedListKind_typ;
	END_VAR
END_FUNCTION

FUNCTION initListSvc : BOOL
	VAR_INPUT
		memValid : BOOL;
	END_VAR
END_FUNCTION

FUNCTION listSvcDeleteCurrentNode : UINT
	VAR_INPUT
		l : linkedList_typ;
	END_VAR
END_FUNCTION

FUNCTION listSvcGetHeadData : UDINT
	VAR_INPUT
		l : linkedList_typ;
	END_VAR
END_FUNCTION

FUNCTION listSvcGetCurrNodeData : UDINT
	VAR_INPUT
		l : linkedList_typ;
	END_VAR
END_FUNCTION

FUNCTION listSvcGetLastNodeData : UDINT
	VAR_INPUT
		l : linkedList_typ;
	END_VAR
END_FUNCTION

FUNCTION listSvcGoNextNodeAndGetData : UDINT
	VAR_INPUT
		l : linkedList_typ;
	END_VAR
END_FUNCTION

FUNCTION listSvcCharListToStringArray : UDINT
	VAR_INPUT
		l : linkedList_typ;
		s : STRING[7];
		sLength : UDINT;
		elements : UDINT;
		offset : UDINT;
		pageOffsetFactor : UDINT;
		maxNodes : UDINT;
		direction : BOOL;
		filterString : STRING[7];
	END_VAR
END_FUNCTION

FUNCTION listCurrentEntries : UDINT
	VAR_INPUT
		l : linkedList_typ;
		a : REFERENCE TO UDINT;
		elements : UDINT;
		offset : UDINT;
		pageOffsetFactor : UDINT;
		getData : BOOL;
	END_VAR
END_FUNCTION
```

#### wbrListSvc.c
```c
/********************************************************************
 * \copyright -- Piedmont Automation
 ********************************************************************
 * Program : wbrListSvc
 * \file :   wbrListSvc.c
 * \author : Blanton Radford
 * \date Created: May 07, 2015
 ******************************************************************* /
 * Implementation of library wbrListSvc
 ********************************************************************/

#ifdef __cplusplus
  extern "C"
  {
#endif

// #include "wbrsprintf_C.h"
#include "wbrListSvc.h"
#include <string.h>

listNode_typ *  head,
             *  curr;

linkedList_typ *   lists;                  //!<  the list of lists

/*! \todo - document the func

 \todo - use 2nd int argument to insert nodes, neg before, pos after, zero adds at head/tail depending on setting
 \todo
*/
static UDINT lsAddNode(linkedList_typ* l, int offset)
{
 listNode_typ * posn                                                            //!<  pointer to node holding the insert position (insert before)
            , * node=   (listNode_typ *) memSvcAllocate(sizeof(listNode_typ))   //!<  new node
            ;

  //! \todo   check private count var lsAddNodeInProcess - should not be needed with queues using dummy tail

  if(node == 0) return  0;
  //! \todo   if(!lsListExists)   return  something meaningful;

  l->numNodes++;

       if(offset < 0){         posn=  l->curr;
                               for( ; offset < 1; offset++)   posn=  posn->prev;
       }
  else if(offset > 0){         posn=  l->curr->next;
                               for( ; offset > 1; offset--)   posn=  posn->next;
       }
  else if(l->kind == lsSTACK)  posn=  l->head;
  else                         posn=  l->dumm;   //  lsQUEUE

  node->next=       posn;
  node->prev=       posn->prev;

  posn->prev->next=  node;
  posn->prev=        node;

  if(l->kind == lsSTACK)
  {
    l->head=  node;
    return  l->head->pData= memSvcAllocate(l->size);
  }

  l->listProcessed= 0;

  return  l->dumm->prev->pData= memSvcAllocate(l->size);    //! \todo   choice to use existing mem for pData
}

/*! \todo

    \todo   choice to use existing mem for pData
            ability to use array as data, e.g. for sorting
            allocate blocks of nodes
*/
UDINT listSvcRequestListNode(linkedList_typ* l)
{
  if((l->head->next == l->dumm) && (l->head->pData == 0))       //  i.e. the list is empty
    return  l->head->pData= memSvcAllocate(l->size);    //! \todo   choice to use existing mem for pData

  return  lsAddNode(l, 0);    //! \todo   choice to use existing mem for pData
}

/*! \todo
*/
// linkedList_typ * listSvcRequestList(UDINT size, linkedListKind_typ kind)
UDINT listSvcRequestList(UDINT size, linkedListKind_typ kind)
{
  linkedList_typ * l=  (linkedList_typ *)listSvcRequestListNode(lists);                                                         //  add new node to p for a new list

  //! \todo   handle alloc err

  l->head=     (listNode_typ *) memSvcAllocate(sizeof(listNode_typ));               //  head is permanent, will not be deleted, but can hold data
  l->dumm=     (listNode_typ *) memSvcAllocate(sizeof(listNode_typ));               //  dumm is a dummy tail.  See documentation for its purpose

  //! \todo   handle alloc errs

  // return  l;                                                         //  DBG:

  l->head->next = l->dumm;
  l->head->prev = l->dumm;

  l->dumm->next=  l->head;
  l->dumm->prev=  l->head;

  l->curr=  l->head;
  // l->dumm=  l->head;                                         //!  \todo  change to support dummy tail and permanent head

  l->size=  size;
  l->kind=  kind;
  l->numNodes= 1;
  l->listProcessed= 1;

  curr=     l->curr;

  return  (UDINT)l;                                                         //
}

/*!
 \warning   this init must be called in the first Init-SP in TC#1
            after memory is initialized
*/
BOOL initListSvc(BOOL memValid)
{
  if(!memValid)   return  0;      //!<  \todo   report error

  head=   (listNode_typ *) memSvcAllocate(sizeof(listNode_typ));                  //  create node for list of lists

  head->pData=   (UDINT)memSvcAllocate(sizeof(linkedList_typ));                   //  create lists list data (header) at pData

  lists=  (linkedList_typ *)head->pData;                                      //  lists is listIdent for the list of lists

  lists->head=   lists->dumm=   lists->curr=  head;                           //  init struct lists' members
  lists->head->next=  lists->head->prev=  lists->head;
  lists->size=  sizeof(linkedList_typ);
  lists->kind=  lsSTACK;

  return  1;
}

UINT listSvcDeleteCurrentNode(linkedList_typ * l)
{
 UINT status;

  if(l->curr == l->dumm)    return  0;

  if(l->curr->pData)
  {
    status= memSvcFree((UDINT)l->curr->pData);
    //! \todo   handle free error, see later in function
    l->curr->pData= 0;
  }
  // else
  // {
    //! \todo   report no mem to free
  // }

  if(l->head->next == l->dumm)
  {
    l->listProcessed= 1;
    return  0;    //! \todo   return status code for attempt to delete permanent head
  }

  l->curr->prev->next=  l->curr->next;
  l->curr->next->prev=  l->curr->prev;

  if(l->curr == l->head)    l->head=  l->curr->next;          //  pop/dequeue if deleting the head

  // curr= l->curr->prev;                        //  This assignment will enable GetNextNode() to function properly
  curr= l->curr->next;                        //  Automatically get next, no need to call GetNextNode()

  status+= memSvcFree((UDINT)l->curr);

  l->curr=  curr;
  l->numNodes--;

  if(status != 0)
  {
    //!   \todo   possibly loop to try again n times?
    //!   \todo   handle error, flag address for later memory cleanup
  }

  return  status;
}

/*! \brief    Returns the head node's data address
              Also points curr to head so that listSvcDeleteCurrentNode() can delete
    \pre      \todo
    \warning  \todo

*/
UDINT listSvcGetHeadData(linkedList_typ * l)
{
  if(!l->head->pData)   return  0;

  l->curr=  l->head;                                          //  allows listSvcDeleteCurrentNode() to delete the head once the head's data is no longer needed

  l->listProcessed= 0;                                        //  Reset for Get****NodeData functions

  return  l->curr->pData;
}

/*! \brief    Returns the current node's data address
    \pre
    \warning  Check that pData has a valid address, e.g. != 0

*/
UDINT listSvcGetLastNodeData(linkedList_typ * l)
{
  return  l->dumm->prev->pData;
}

/*! \brief    Returns the current node's data address
    \pre
    \warning  Check that pData has a valid address, e.g. != 0

*/
UDINT listSvcGetCurrNodeData(linkedList_typ * l)
{
  return  l->curr->pData;
}

/*! \brief    Advances to the next node and returns the data address
              This function has special conditions for the head and dumm nodes
    \pre      \todo
    \warning  \todo

*/
UDINT listSvcGoNextNodeAndGetData(linkedList_typ * l)
{
  if(l->curr == l->head)  l->listProcessed= 0;

  curr=   l->curr=  l->curr->next;

  if(l->curr == l->dumm)
  {
    curr= l->curr=  l->head;
    l->listProcessed= 1;
  }

  return  l->curr->pData;
}

/*! \brief    Print list of char strings to string array

    \pre      An array of sufficient size to contain all strings of interest
    \warning  \todo
    \todo     Provide an index that will allow <elements> nodes to be listed starting at the index
              Allow paging by offsetting <index> by <elements> * <offsetFactor>
                Possibly show a full page if pages > 1 and the end of the list is reached
              Begin destroying nodes when memInfo.maxBlockSizeFree == tbd% of configured memory block size
                This is needed since this func is used for logging to prevent the logging from growing forever
              Option to save list to file when above todo is triggered
                Option to save list on request
              Use wbrListSvcStringList_typ as input

**********************************************/
UDINT listSvcCharListToStringArray(

            linkedList_typ * l        //!<  The list to be read into a string array
          , char* s                   //!<  Pointer to the string array used for viewing
          , UDINT sLength             //!<  Length of the strings
          , UDINT elements            //!<  Number of elements in the array
          , UDINT offset              //!<  Offset into the list
          , UDINT pageOffsetFactor    //!<  Additional offset into the list by n "pages" of size <elements>
          , UDINT maxNodes            //!<  Maximum number of nodes to keep in the list.  Can be less than elements.  Zero will allow unlimited nodes.
          , BOOL  direction           //!<  Direction the list is read.  See code comments for details
          , char* filterString        //!<  String used to filter the list.  Any node data which the first chars don't match will not be added to the view list.
          )

// ****************************************** /
{
 UDINT      i
          , o
          , elementsPrinted=  0
          , elementsCleared=  0
          , nodesSkipped=     0
          , nodesProcessed=   0
          , order=  (l->kind << 1) + direction
          ;

 listNode_typ * work= l->dumm;

  offset+=  pageOffsetFactor * elements;
  o=  offset;

  if(offset >= l->numNodes)  {
    wbrsnprintf(s, sLength, "Offset too large.  Nothing to print.");
    s+= sLength;
    for(i=  1;  i < elements ; i++, s+= sLength)
      s[0]= 0;
    return  1;
  }

  for(i=  0;  (elementsPrinted + elementsCleared) < elements ; i++)
  {
    nodesProcessed=  elementsPrinted + elementsCleared + nodesSkipped;

    switch(order)
    {
     case   0:      //  stack, FIFO   lsPRINT_CHAR_STACK_FIFO
     case   3:      //  queue, LIFO   lsPRINT_CHAR_QUEUE_LIFO
      if(maxNodes && l->numNodes > maxNodes)
      {
        l->curr=  work->next;
        while(l->numNodes > maxNodes)  {
          listSvcDeleteCurrentNode(l);
        }
      }

      while(o > 0)  work= work->prev, o--, nodesSkipped++;

      if(work->prev == l->dumm)   {
        s[0]= 0;
        elementsCleared++;
        s+= sLength;
        continue;
      }

      work= work->prev;

      break;

     case   1:      //  stack, LIFO   lsPRINT_CHAR_STACK_LIFO
     case   2:      //  queue, FIFO   lsPRINT_CHAR_QUEUE_FIFO
      if(maxNodes && l->numNodes > maxNodes)
      {
        l->curr=  work->prev;
        while(l->numNodes > maxNodes)  {
          listSvcDeleteCurrentNode(l);
          if(l->curr->prev != l->dumm)
            l->curr=  l->curr->prev;
        }
      }

      while(o > 0)  work= work->next, o--, nodesSkipped++;

      if(work->next == l->dumm)  {
        s[0]= 0;
        elementsCleared++;
        s+= sLength;
        continue;
      }

      work= work->next;
      break;
    }

    if(!work->pData)                        return  elementsPrinted;
    if(strncmp((char *)work->pData, filterString, strlen(filterString)))  {
      nodesSkipped++;
      continue;
    }

    elementsPrinted++;
    // wbrsnprintf(s, sLength, "%s", (char *)work->pData);
    // wbrsnprintf(s, sLength, "%d. %s"
              // , (elementsPrinted + offset)
              // , (char *)work->pData
             // );
    wbrsnprintf(s, sLength, "%*d. %s"
              , (elements + offset) > 99 ? 3 : 2
              , (elementsPrinted + offset)
              , (char *)work->pData
             );
    s+= sLength;
  }

  return  elementsPrinted;
}

/*! \brief    List node addresses for debugging

    \pre      An array of sufficient size to contain all addresses of interest
    \warning  \todo
    \todo     Provide an index that will allow <elements> nodes to be listed starting at the index
              Allow paging by offsetting <index> by <elements> * <offsetFactor>
              Possibly combine this with listSvcCharListToStringArray() since the code is similar.
                This will require moving this func above listSvcCharListToStringArray().

**********************************************/
UDINT listCurrentEntries(

            linkedList_typ * l        //!<  the list to be read into an array
          , UDINT a[]                 //!<  the array
          , UDINT elements            //!<  number of elements in the array
          , UDINT offset              //!<  offset into the list
          , UDINT pageOffsetFactor    //!<  additional offset into the list by n "pages" of size <elements>
          , BOOL  getData             //!<  if TRUE, get the address of the data.  Else, get the node address
          )

// ****************************************** /
{
 UDINT          i;

 listNode_typ * work=  l->head;

  offset+=  pageOffsetFactor * elements;

  for(  ;  offset > 0; work= work->next, offset--)     {  }

  for(i= 0; i<elements ; work= work->next, i++)
  {
    if(getData)   a[i]= (UDINT)work->pData;               //
    else          a[i]= (UDINT)work;               //
    if(work->next == l->dumm)  break;
  }

  if(i < (elements - 1))    a[++i]=  0;

  return  i;
}

#ifdef __cplusplus
  }
#endif
```

### Library Logical/UserLibraries/wbrServices/wbrPingSvc

#### wbrPingSvc.typ
```iecst
(*** /*****************************************************************
 * \copyright -- Piedmont Automation
 ********************************************************************
 * Program : wbrPingSvc
 * \file :   wbrPingSvc.typ
 * \author : Blanton Radford
 * \date Created: June 22, 2015
 ********************************************************************
 * Data types of library wbrPingSvc
 ****************************************************************/ ****)

TYPE
	wbrPingService_typ : 	STRUCT
		fb : IcmpPing; (*Ping function block*)
		enable : BOOL; (*optional enable can be used to call function only when desired*)
		timeout : UINT := 100; (*Multiply by 10ms*)
		count : UINT := 0;
		errorStatus : UINT := 0;
		failed : BOOL := FALSE;
		successesToCount : USINT := 4;
		failuresToCount : USINT;
		message1 : STRING[127] := 'No ping tried';
		message : STRING[127] := 'No ping tried';
		logbookID : UDINT; (*Ident of the logbook to log the ping messages to*)
		destIPPrev : STRING[15];
		destIPAddr : STRING[15] := '192.168.44.220';
		repeatTime : UINT := 1000; (*Multiply by 1ms*)
		retryTimer : TON;
	END_STRUCT;
END_TYPE
```

#### wbrPingSvc.fun
```iecst
(********************************************************************
 * COPYRIGHT -- Piedmont Automation
 ********************************************************************
 * Library: wbrPingSvc
 * File: wbrPingSvc.fun
 * Author: Blanton Radford
 * Created: June 22, 2015
 ********************************************************************
 * Functions and function blocks of library wbrPingSvc
 ********************************************************************)

FUNCTION wbrPingSvcInit : DINT
	VAR_INPUT
		p : wbrPingService_typ;
	END_VAR
END_FUNCTION

FUNCTION wbrPingStation : DINT
	VAR_INPUT
		p : wbrPingService_typ;
	END_VAR
END_FUNCTION

FUNCTION wbrSQL_DT2_ISOFmtdStringFromDT : DINT
	VAR_INPUT
		pDT : DTStructure;
		pDst : STRING[31];
		dstSize : UDINT;
	END_VAR
END_FUNCTION
```
